# B&R Automation Studio project SDCAxis
Automation Studio 4.5.2.102; Default project; technology packages: Acp10Arnc0 1.0.0

## Configuration Real

CPU 4PP065.0571-P74, AutomationRuntime D4.52, Build 4.1.2, Vc V4.25.0, Safety 1.6

### Task classes (Cpu.sw)
```
Cyclic#1 (cycle 2000 us, tolerance 0 us):
  SDCAxisCtr <- SDCAxisCtrl_X.prg
  SDCAxisCt2 <- SDCAxisCtrl_Z.prg
  SDCAxisCt1 <- SDCAxisCtrl_Y.prg
DataObjects: Arnc0sys
NcDataObjects: AxisInit <- AxisInit.dob, gAxis05a <- gAxis05obj.gAxis05a.dob, gAxis03a <- gAxis03obj.gAxis03a.dob, AxisApt <- AxisApt.dob, gAxis05i <- gAxis05obj.gAxis05i.dob, gAxis03i <- gAxis03obj.gAxis03i.dob, CncInit <- CncInit.dob, CncProg <- CncProg.dob, gmcipvar <- GmcIpUserConfig.gmcipvar.dob, gmcipfun <- GmcIpUserConfig.gmcipfun.dob, gmcipfub <- GmcIpUserConfig.gmcipfub.dob, gmcipubr <- GmcIpUserConfig.gmcipubr.dob, gmcipusm <- GmcIpUserConfig.gmcipusm.dob, gmcipui <- GmcIpUserConfig.gmcipui.dob, gmcipus <- GmcIpUserConfig.gmcipus.dob, gmcipuc <- GmcIpUserConfig.gmcipuc.dob, gmcipsys <- GmcIpConfig.gmcipsys.dob, gmciplbr <- GmcIpConfig.gmciplbr.dob, gmcipcbr <- GmcIpConfig.gmcipcbr.dob, gmciplsm <- GmcIpConfig.gmciplsm.dob, gmcipcsm <- GmcIpConfig.gmcipcsm.dob, gmcipcfg <- GmcIpConfig.gmcipcfg.dob, gmcipiec <- GmcIpConfig.gmcipiec.dob, gmciplog <- GmcIpConfig.gmciplog.dob, gmcipesm <- GmcIpConfig.gmcipesm.dob, gmcipmxd <- GmcIpConfig.gmcipmxd.dob, gmcipmx <- GmcIpConfig.gmcipmx.dob
Binaries: TCData, udbdef, ashwac, ashwd, asfw, iomap, sysconf, Role, User, arconfig, Arnc0map, arnc0cfg, Acp10map, acp10cfg, Acp10map1
Libraries: Acp10sdc, Library, Acp10man, Acp10_MC, sys_lib, brsystem, asstring, AsMath, Arnc0man, DataObj, AsArLog, FileIO, AsArProf, AsMem, Runtime, astime, Acp10par, NcGlobal, powerlnk, asiotime, asieccon
```

### Hardware
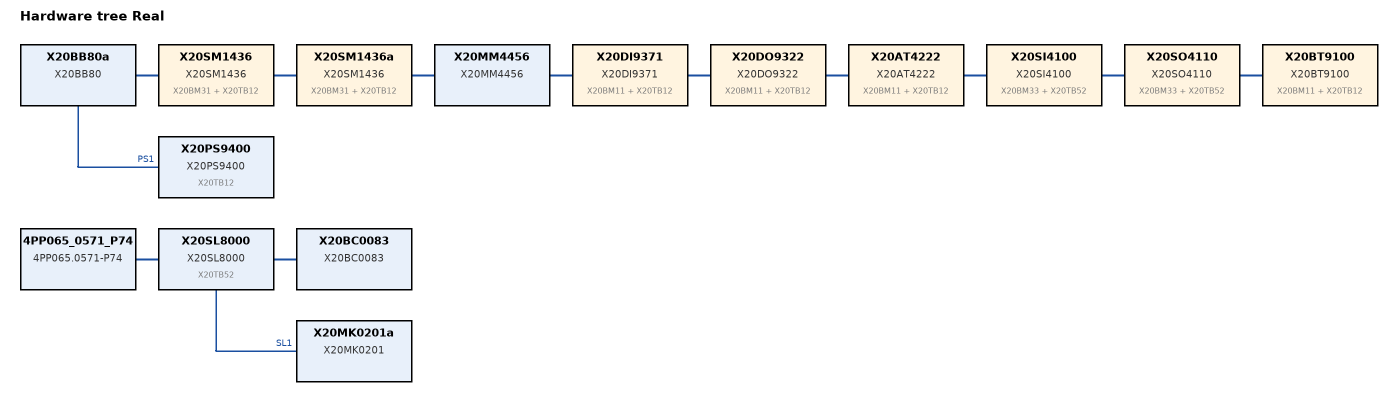
```
4PP065_0571_P74 : 4PP065.0571-P74 v1.1.2.0
  Connector IF4:
    EplInterfaceRedundant = 0
    EplEthInterfaceRedundant = 0
  Connector IF5:
    ActivateDevice = 1
    Mode = Manual
    InternetAddress = 10.0.1.14
    SubnetMask = 255.255.255.0
  ConfigurationID = labBR
  TimerDeviceType = EPLX2X
  TimerDevice = 4PP065_0571_P74.IF4
  TaskClassIdleTime = 2000
  Cyclic1Duration = 2000
  Cyclic1Tolerance = 0
  Cyclic1Output = 1
  Cyclic3Tolerance = 0
  VcObjectName = Visu
X20AT4222 : X20AT4222 v1.2.3.0  [SS1 -> X20TB12f.SS; SL -> X20BM11c.SL1]
X20BB80a : X20BB80 v1.0.2.0
X20BC0083 : X20BC0083 v2.7.0.0  [PLK1 -> X20SL8000.PLK2 (NodeNumber=2) [Cable Type=PowerlinkCable, Length=10, Version=1.0.0.2]; SL -> X20BB80a.SL1]
X20BM11a : X20BM11 v1.0.0.1  [X2X1 -> X20MM4456.X2X2]
X20BM11b : X20BM11 v1.0.0.1  [X2X1 -> X20BM11a.X2X2]
X20BM11c : X20BM11 v1.0.0.1  [X2X1 -> X20BM11b.X2X2]
X20BM11d : X20BM11 v1.0.0.1  [X2X1 -> X20BM33b.X2X2]
X20BM31a : X20BM31 v1.0.0.1  [X2X1 -> X20BB80a.IF1]
X20BM31b : X20BM31 v1.0.0.1  [X2X1 -> X20BM31a.X2X2]
X20BM33a : X20BM33 v1.0.0.4  [X2X1 -> X20BM11c.X2X2]
X20BM33b : X20BM33 v1.0.0.4  [X2X1 -> X20BM33a.X2X2]
X20BT9100 : X20BT9100 v1.0.3.0  [SS1 -> X20TB12g.SS; SL -> X20BM11d.SL1]
X20DI9371 : X20DI9371 v1.0.2.0  [SS1 -> X20TB12d.SS; SL -> X20BM11a.SL1]
X20DO9322 : X20DO9322 v1.0.3.0  [SS1 -> X20TB12e.SS; SL -> X20BM11b.SL1]
X20MK0201a : X20MK0201 v1.0.0.0  [SL -> X20SL8000.SL1]
X20MM4456 : X20MM4456 v1.1.5.0  [X2X1 -> X20BM31b.X2X2]
X20PS9400 : X20PS9400 v1.0.2.4  [SS1 -> X20TB12b.SS; PS -> X20BB80a.PS1]
X20SI4100 : X20SI4100 v1.10.1.1  [SS1 -> X20TB52b.SS; SL -> X20BM33a.SL1]
X20SL8000 : X20SL8000 v1.6.5.1  [PLK1 -> 4PP065_0571_P74.IF4 (NodeNumber=1) [Cable Type=PowerlinkCable, Length=10, Version=1.0.0.2]; PLK2 -> X20BC0083.PLK1 (NodeNumber=1) [Cable Type=PowerlinkCable, Length=10, Version=1.0.0.2]; SS1 -> X20TB52a.SS]
  SafeProject = SafeLOGIC-1
X20SM1436 : X20SM1436 v1.4.2.1  [SS1 -> X20TB12a.SS; SL -> X20BM31a.SL1]
X20SM1436a : X20SM1436 v1.4.2.1  [SS1 -> X20TB12c.SS; SL -> X20BM31b.SL1]
X20SO4110 : X20SO4110 v1.10.1.1  [SS1 -> X20TB52c.SS; SL -> X20BM33b.SL1]
  SafeLogicID = 2
  SafeModuleID = 3
X20TB12a : X20TB12 v1.0.0.0
X20TB12b : X20TB12 v1.0.0.0
X20TB12c : X20TB12 v1.0.0.0
X20TB12d : X20TB12 v1.0.0.0
X20TB12e : X20TB12 v1.0.0.0
X20TB12f : X20TB12 v1.0.0.0
X20TB12g : X20TB12 v1.0.0.0
X20TB52a : X20TB52 v1.0.0.1
X20TB52b : X20TB52 v1.0.0.1
X20TB52c : X20TB52 v1.0.0.1
```

### IoMap.iom - 4PP065_0571_P74/IoMap.iom
```iecst
VAR_CONFIG
	::SDCAxisCtr:pwm_period AT %QW."X20MM4456".PeriodDurationPWM;
	::SDCAxisCtr:coil_pwm_value AT %QW."X20MM4456".PulseWidthCurrentPWM04;
	::SDCAxisCtr:axis_X.pwm_value AT %QW."X20MM4456".PulseWidthCurrentPWM01;
	::SDCAxisCtr:axis_X.reset_error AT %QX."X20MM4456".ClearError01;
	::SDCAxisCtr:axis_X.reset_counter AT %QX."X20MM4456".ResetCounter01;
	::SDCAxisCtr:axis_X.counter AT %IW."X20MM4456".Counter01;
	::SDCAxisCtr:axis_X.endswitch_a_reached AT %IX."X20MM4456".StatusInput03;
	::SDCAxisCtr:axis_X.endswitch_b_reached AT %IX."X20MM4456".StatusInput04;
	::SDCAxisCtr:coil_powered_X AT %IX."X20DI9371".DigitalInput02;
	::SDCAxisCt1:coil_powered_Y AT %IX."X20DI9371".DigitalInput03;
	::SDCAxisCt2:coil_powered_Z AT %IX."X20DI9371".DigitalInput04;
	::SDCAxisCt1:gaxis03.pwm_value AT %QW."X20MM4456".PulseWidthCurrentPWM02;
	::SDCAxisCt1:gaxis03.reset_error AT %QX."X20MM4456".ClearError02;
	::SDCAxisCt1:gaxis03.reset_counter AT %QX."X20MM4456".ResetCounter02;
	::SDCAxisCt1:gaxis03.counter AT %IW."X20MM4456".Counter02;
	::SDCAxisCt1:gaxis03.endswitch_a_reached AT %IX."X20MM4456".StatusInput07;
	::SDCAxisCt1:gaxis03.endswitch_b_reached AT %IX."X20MM4456".StatusInput08;
	::SDCAxisCt2:gaxis05.pwm_value AT %QW."X20MM4456".PulseWidthCurrentPWM03;
	::SDCAxisCt2:gaxis05.reset_error AT %QX."X20MM4456".ClearError03;
	::SDCAxisCt2:gaxis05.reset_counter AT %QX."X20MM4456".ResetCounter03;
	::SDCAxisCt2:gaxis05.counter AT %IW."X20MM4456".Counter03;
	::SDCAxisCt2:gaxis05.endswitch_a_reached AT %IX."X20MM4456".StatusInput11;
	::SDCAxisCt2:gaxis05.endswitch_b_reached AT %IX."X20MM4456".StatusInput12;
END_VAR
```

### Acp10cfg.ncc - 4PP065_0571_P74/Motion/Acp10cfg.ncc
```
NcConfiguration (Version=3.13.1, NcSwId=Acp10)
  ACP10CF1_typ:
    cnt_nettrc_rec_drive = 1500
    bufsize_trace_upload = 1200
    tc_nc_man_task = Cyclic #1
    glob_pv_as_ncobject = Yes
    ncsys_dl_broadcast = Yes
    ncsys_dl_acp_reset = Yes
    safemc_log_err_to_ax = Yes
    network_init:
      ncsw_init_execute = Yes
      automatic_execute = No
      node_nr_warning = Yes
      net_err_before_ncact = Yes
    nettrc:
      enter_parsecrec = Yes
      enter_ncaction = Yes
      save_ring_startidx = Yes
    cam_prof_download:
      cam_dat_dl_parallel = No
      tc_cam_dl_parallel = Task class for NC Manager task
    sdc_if[0]:
      if_name = SDC_IF1
      mc_broadcast_size = 800
      mc_broadcast_extdat = No
```

### Acp10map.ncm - 4PP065_0571_P74/Motion/Acp10map.ncm
```
NcMapping (NcSwId=Acp10, DisabledNodesAreHidden=False)
```

### Acp10map1.ncm - 4PP065_0571_P74/Motion/Acp10map1.ncm
```
NcMapping (NcSwId=ACP10, DisabledNodesAreHidden=False)
  NcObject AxisX (ModuleAddress=SDC_IF1.ST1, InterfaceType=SDC, Type=ncAXIS, Channel=1, AcoposSimulation=Off, InitParameter=AxisInit, AcoposParameter=gAxis03a, AdditionalData=CNC_Enabled="1" , Disabled=FALSE, ModuleDisabled=FALSE)
  NcObject gAxis03 (ModuleAddress=SDC_IF1.ST2, InterfaceType=SDC, Type=ncAXIS, Channel=1, AcoposSimulation=Off, InitParameter=AxisInit, AcoposParameter=gAxis03a, AdditionalData=CNC_Enabled="1", Disabled=FALSE)
  NcObject gAxis05 (ModuleAddress=SDC_IF1.ST3, InterfaceType=SDC, Type=ncAXIS, Channel=1, AcoposSimulation=Off, InitParameter=AxisInit, AcoposParameter=gAxis03a, AdditionalData=CNC_Enabled="1" , Disabled=FALSE)
```

### Arnc0cfg.ncc - 4PP065_0571_P74/Motion/Arnc0cfg.ncc
```
NcConfiguration (Version=3.13.0, NcSwId=Arnc0)
  ARNC0CFG_typ:
    sampling_rate = 2000
    cnt_nettrc_rec_drive = 150
    bufsize_sys_trace = 16#00005000
    enable_mp_log = Yes
    tc_nc_man_task = Cyclic #1
    bg_load = 1
    glob_pv_as_ncobject = Yes
```

### Arnc0map.ncm - 4PP065_0571_P74/Motion/Arnc0map.ncm
```
NcMapping (NcSwId=Arnc0, DisabledNodesAreHidden=True)
  NcObject CNCsys (Type=ncCNCSYS, Channel=1, AcoposSimulation=Off, InitParameter=CncInit, Disabled=FALSE, ModuleDisabled=FALSE)
  NcObject CNC2 (Type=ncCNCSYS, Channel=2, AcoposSimulation=Off, Disabled=TRUE, ModuleDisabled=FALSE)
  NcObject CNC3 (Type=ncCNCSYS, Channel=3, AcoposSimulation=Off, Disabled=TRUE, ModuleDisabled=FALSE)
  NcObject CNC4 (Type=ncCNCSYS, Channel=4, AcoposSimulation=Off, Disabled=TRUE, ModuleDisabled=FALSE)
  NcObject CNC5 (Type=ncCNCSYS, Channel=5, AcoposSimulation=Off, Disabled=TRUE, ModuleDisabled=FALSE)
  NcObject CNC6 (Type=ncCNCSYS, Channel=6, AcoposSimulation=Off, Disabled=TRUE, ModuleDisabled=FALSE)
  NcObject CNC7 (Type=ncCNCSYS, Channel=7, AcoposSimulation=Off, Disabled=TRUE, ModuleDisabled=FALSE)
  NcObject CNC8 (Type=ncCNCSYS, Channel=8, AcoposSimulation=Off, Disabled=TRUE, ModuleDisabled=FALSE)
  NcObject CNC9 (Type=ncCNCSYS, Channel=9, AcoposSimulation=Off, Disabled=TRUE, ModuleDisabled=FALSE)
  NcObject CNC10 (Type=ncCNCSYS, Channel=10, AcoposSimulation=Off, Disabled=TRUE, ModuleDisabled=FALSE)
  NcObject CNC11 (Type=ncCNCSYS, Channel=11, AcoposSimulation=Off, Disabled=TRUE, ModuleDisabled=FALSE)
  NcObject CNC12 (Type=ncCNCSYS, Channel=12, AcoposSimulation=Off, Disabled=TRUE, ModuleDisabled=FALSE)
  NcObject CNC13 (Type=ncCNCSYS, Channel=13, AcoposSimulation=Off, Disabled=TRUE, ModuleDisabled=FALSE)
  NcObject CNC14 (Type=ncCNCSYS, Channel=14, AcoposSimulation=Off, Disabled=TRUE, ModuleDisabled=FALSE)
  NcObject CNC15 (Type=ncCNCSYS, Channel=15, AcoposSimulation=Off, Disabled=TRUE, ModuleDisabled=FALSE)
  NcObject CNC16 (Type=ncCNCSYS, Channel=16, AcoposSimulation=Off, Disabled=TRUE, ModuleDisabled=FALSE)
  NcObject CNC17 (Type=ncCNCSYS, Channel=17, AcoposSimulation=Off, Disabled=TRUE, ModuleDisabled=FALSE)
  NcObject CNC18 (Type=ncCNCSYS, Channel=18, AcoposSimulation=Off, Disabled=TRUE, ModuleDisabled=FALSE)
  NcObject CNC19 (Type=ncCNCSYS, Channel=19, AcoposSimulation=Off, Disabled=TRUE, ModuleDisabled=FALSE)
  NcObject CNC20 (Type=ncCNCSYS, Channel=20, AcoposSimulation=Off, Disabled=TRUE, ModuleDisabled=FALSE)
  NcObject CNC21 (Type=ncCNCSYS, Channel=21, AcoposSimulation=Off, Disabled=TRUE, ModuleDisabled=FALSE)
  NcObject CNC22 (Type=ncCNCSYS, Channel=22, AcoposSimulation=Off, Disabled=TRUE, ModuleDisabled=FALSE)
  NcObject CNC23 (Type=ncCNCSYS, Channel=23, AcoposSimulation=Off, Disabled=TRUE, ModuleDisabled=FALSE)
  NcObject CNC24 (Type=ncCNCSYS, Channel=24, AcoposSimulation=Off, Disabled=TRUE, ModuleDisabled=FALSE)
```

## Configuration Simulation

CPU , AutomationRuntime J4.25, Safety 1.10

### Task classes (Cpu.sw)
```
Cyclic#1 (cycle 2000 us, tolerance 0 us):
  SDCAxisCtr <- SDCAxisCtrl_X.prg
  ncsdcctrl <- ncsdcctrl.prg
DataObjects: Acp10sys
NcDataObjects: AxisApt <- AxisApt.dob, AxisInit <- AxisInit.dob, acp10etxen <- acp10etxen.dob, gAxis05a <- gAxis05obj.gAxis05a.dob, gAxis05i <- gAxis05obj.gAxis05i.dob
Binaries: TCData, ashwd, sysconf, asfw, arconfig, iomap, Acp10map, Acp10map1, arnc0cfg, acp10cfg
Libraries: AsIecCon, astime, Acp10sdc, Acp10man, Acp10par, NcGlobal, asstring, AsIOTime, Acp10_MC, brsystem, sys_lib, Runtime, Acp10sim, fileio, powerlnk, Library, AsBrStr
```

### Hardware
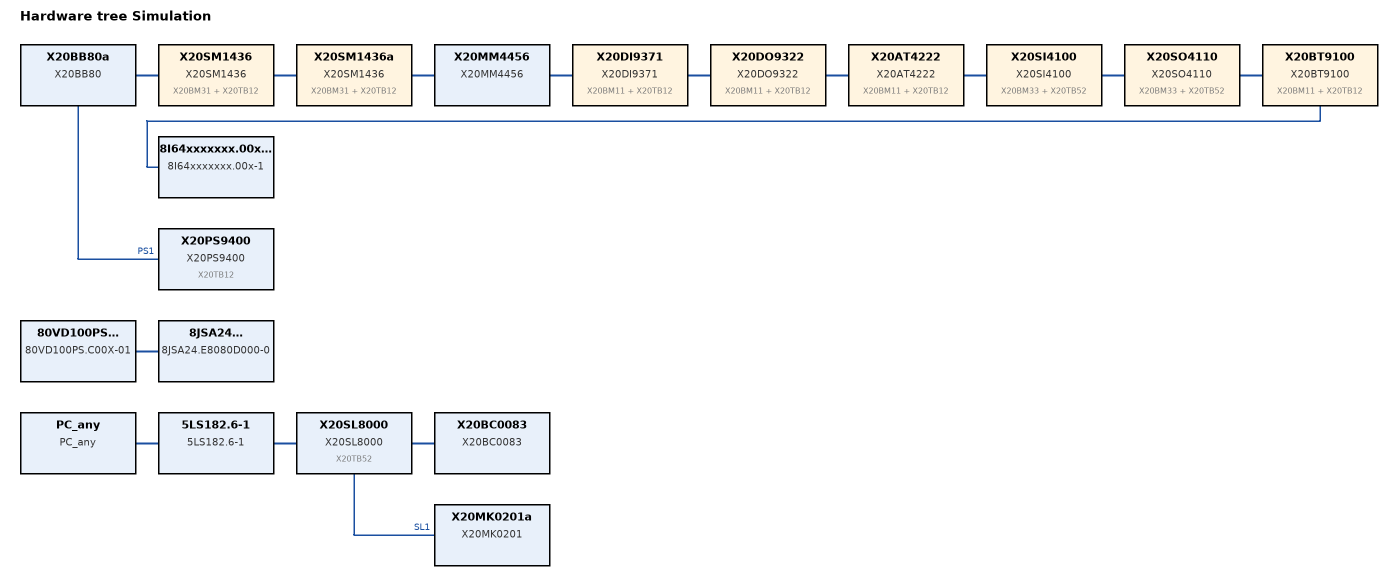
```
5LS182.6-1 : 5LS182.6-1 v1.3.0.0  [SL -> PC_any.SL1]
80VD100PS.C00X-01 : 80VD100PS.C00X-01 v2.3.0.1
8I64xxxxxxx.00x-1 : 8I64xxxxxxx.00x-1 v1.3.9.1  [X2X1 -> X20BT9100.X2X1 [Cable Type=X2XCable, Length=10, Version=1.0.0.2]]
  BothEndSwitchesAreNormallyOpen_r1 = on
  QuickStopIsNormallyOpen_r1 = on
8JSA24.E8080D000-0 : 8JSA24.E8080D000-0 v1.0.6.30  [MT -> 80VD100PS.C00X-01.MT1]
PC_any : PC_any v1.1.0.0 (OrderNumber=PC)
  ConfigurationID = SDCAxis_Simulation
  SystemTick = 2000
  Cyclic1Duration = 2000
  Cyclic1Tolerance = 0
  Cyclic1Output = 1
X20AT4222 : X20AT4222 v1.2.3.0  [SS1 -> X20TB12f.SS; SL -> X20BM11c.SL1]
X20BB80a : X20BB80 v1.0.2.0
X20BC0083 : X20BC0083 v2.7.0.0  [PLK2 -> X20SL8000.PLK2 (NodeNumber=2) [Cable Type=PowerlinkCable, Length=10, Version=1.0.0.2]; SL -> X20BB80a.SL1]
X20BM11a : X20BM11 v1.0.0.1  [X2X1 -> X20MM4456.X2X2]
X20BM11b : X20BM11 v1.0.0.1  [X2X1 -> X20BM11a.X2X2]
X20BM11c : X20BM11 v1.0.0.1  [X2X1 -> X20BM11b.X2X2]
X20BM11d : X20BM11 v1.0.0.1  [X2X1 -> X20BM33b.X2X2]
X20BM31a : X20BM31 v1.0.0.1  [X2X1 -> X20BB80a.IF1]
X20BM31b : X20BM31 v1.0.0.1  [X2X1 -> X20BM31a.X2X2]
X20BM33a : X20BM33 v1.0.0.4  [X2X1 -> X20BM11c.X2X2]
X20BM33b : X20BM33 v1.0.0.4  [X2X1 -> X20BM33a.X2X2]
X20BT9100 : X20BT9100 v1.0.3.0  [SS1 -> X20TB12g.SS; SL -> X20BM11d.SL1]
X20DI9371 : X20DI9371 v1.0.2.0  [SS1 -> X20TB12d.SS; SL -> X20BM11a.SL1]
X20DO9322 : X20DO9322 v1.0.3.0  [SS1 -> X20TB12e.SS; SL -> X20BM11b.SL1]
X20MK0201a : X20MK0201 v1.0.0.0  [SL -> X20SL8000.SL1]
X20MM4456 : X20MM4456 v1.1.5.0  [X2X1 -> X20BM31b.X2X2]
X20PS9400 : X20PS9400 v1.0.2.4  [SS1 -> X20TB12b.SS; PS -> X20BB80a.PS1]
X20SI4100 : X20SI4100 v1.10.1.1  [SS1 -> X20TB52b.SS; SL -> X20BM33a.SL1]
X20SL8000 : X20SL8000 v1.6.5.1  [PLK1 -> 5LS182.6-1.IF1 (NodeNumber=1) [Cable Type=PowerlinkCable, Length=10, Version=1.0.0.2]; PLK2 -> X20BC0083.PLK2 (NodeNumber=1) [Cable Type=PowerlinkCable, Length=10, Version=1.0.0.2]; SS1 -> X20TB52a.SS]
  SafeProject = SafeLOGIC-1
X20SM1436 : X20SM1436 v1.4.2.1  [SS1 -> X20TB12a.SS; SL -> X20BM31a.SL1]
X20SM1436a : X20SM1436 v1.4.2.1  [SS1 -> X20TB12c.SS; SL -> X20BM31b.SL1]
X20SO4110 : X20SO4110 v1.10.1.1  [SS1 -> X20TB52c.SS; SL -> X20BM33b.SL1]
  SafeLogicID = 2
  SafeModuleID = 3
X20TB12a : X20TB12 v1.0.0.0
X20TB12b : X20TB12 v1.0.0.0
X20TB12c : X20TB12 v1.0.0.0
X20TB12d : X20TB12 v1.0.0.0
X20TB12e : X20TB12 v1.0.0.0
X20TB12f : X20TB12 v1.0.0.0
X20TB12g : X20TB12 v1.0.0.0
X20TB52a : X20TB52 v1.0.0.1
X20TB52b : X20TB52 v1.0.0.1
X20TB52c : X20TB52 v1.0.0.1
```

### IOMap.iom - PC_any/IOMap.iom
```iecst
VAR_CONFIG
	::SDCAxisCtr:pwm_period AT %QW."X20MM4456".PeriodDurationPWM;
	::SDCAxisCtr:coil_pwm_value AT %QW."X20MM4456".PulseWidthCurrentPWM04;
	::SDCAxisCtr:axis_X.pwm_value AT %QW."X20MM4456".PulseWidthCurrentPWM01;
	::SDCAxisCtr:axis_X.reset_error AT %QX."X20MM4456".ClearError01;
	::SDCAxisCtr:axis_X.reset_counter AT %QX."X20MM4456".ResetCounter01;
	::SDCAxisCtr:axis_X.counter AT %IW."X20MM4456".Counter01;
	::SDCAxisCtr:axis_X.endswitch_a_reached AT %IX."X20MM4456".StatusInput03; (*Logical condition input 01=Motor 01:A*)
	::SDCAxisCtr:axis_X.endswitch_b_reached AT %IX."X20MM4456".StatusInput04; (*Logical condition input 02=Motor 01:B*)
	::SDCAxisCtr:coil_powered AT %IX."X20DI9371".DigitalInput01;
	Cyclic#1.gAxis03_DrvIf.iLifeCnt AT %IB."8I64xxxxxxx.00x-1".SDC_LifeCnt;
	Cyclic#1.gAxis03_DrvIf.iDrvOK AT %IX."8I64xxxxxxx.00x-1".ETAD_Input_Bool_02;
	Cyclic#1.gAxis03_DrvIf.oSetTime AT %QW."8I64xxxxxxx.00x-1".SDC_SetTime;
	Cyclic#1.gAxis03_DrvIf.oSetPos AT %QW."8I64xxxxxxx.00x-1".LFRD_Output;
	Cyclic#1.gAxis03_DiDoIf.iLifeCntDriveReady AT %IB."8I64xxxxxxx.00x-1".SDC_LifeCnt;
	Cyclic#1.gAxis03_DiDoIf.iLifeCntDriveEnable AT %IB."8I64xxxxxxx.00x-1".SDC_LifeCnt;
	Cyclic#1.gAxis03_DiDoIf.oDriveEnable AT %QX."8I64xxxxxxx.00x-1".CMDD_Output_Bool_00;
	Cyclic#1.gAxis03_ModuleOk AT %QX."8I64xxxxxxx.00x-1".CMDD_Output_Bool_01;
	Cyclic#1.gAxis03_ModuleOk AT %QX."8I64xxxxxxx.00x-1".CMDD_Output_Bool_02;
	Cyclic#1.gAxis03_ModuleOk AT %IX."8I64xxxxxxx.00x-1".ModuleOk;
	Cyclic#1.gAxis03_DiDoIf.oDriveEnable AT %QX."8I64xxxxxxx.00x-1".CMDD_Output_Bool_03;
	Cyclic#1.gAxis03_DiDoIf.iDriveReady AT %IX."8I64xxxxxxx.00x-1".ETAD_Input_Bool_02;
	      Cyclic#1.gAxis05_DrvIf.iLifeCnt AT %IB."X20SM1436".LifeCnt;
	      Cyclic#1.gAxis05_DrvIf.iDrvOK AT %IX."X20SM1436".DrvOk01;
	      Cyclic#1.gAxis05_DrvIf.oBoostCurrent AT %QX."X20SM1436".BoostCurrent01;
	      Cyclic#1.gAxis05_DrvIf.oStandStillCurrent AT %QX."X20SM1436".StandstillCurrent01;
	      Cyclic#1.gAxis05_DrvIf.oSetTime AT %QW."X20SM1436".SetTime01;
	      Cyclic#1.gAxis05_MotorStep0 AT %QW."X20SM1436".Motor1Step0;
	      Cyclic#1.gAxis05_DiDoIf.iLifeCntDriveEnable AT %IB."X20SM1436".LifeCnt;
	      Cyclic#1.gAxis05_DiDoIf.iLifeCntDriveReady AT %IB."X20SM1436".LifeCnt;
	      Cyclic#1.gAxis05_DiDoIf.iDriveReady AT %IX."X20SM1436".DrvOk01;
	      Cyclic#1.gAxis05_DiDoIf.oDriveEnable AT %QX."X20SM1436".DriveEnable01;
	      Cyclic#1.gAxis05_EncIf1.iLifeCnt AT %IB."X20SM1436".LifeCnt;
	      Cyclic#1.gAxis05_EncIf1.iEncOK AT %IX."X20SM1436".EncOk01;
	      Cyclic#1.gAxis05_EncIf1.iActPos AT %IW."X20SM1436".ActPos01;
	      Cyclic#1.gAxis05_EncIf1.iRefPulsePos AT %IW."X20SM1436".RefPulsePos01;
	      Cyclic#1.gAxis05_EncIf1.iRefPulseCnt AT %IB."X20SM1436".RefPulseCnt01;
	      Cyclic#1.gAxis05_EncIf1.iActTime AT %IW."X20SM1436".ActTime01;
END_VAR
```

### Acp10cfg.ncc - PC_any/Motion/Acp10cfg.ncc
```
NcConfiguration (Version=3.13.1, NcSwId=Acp10)
  ACP10CF1_typ:
    cnt_nettrc_rec_drive = 150
    bufsize_trace_upload = 1200
    tc_nc_man_task = Cyclic #1
    glob_pv_as_ncobject = Yes
    ncsys_dl_broadcast = Yes
    ncsys_dl_acp_reset = Yes
    safemc_log_err_to_ax = Yes
    network_init:
      ncsw_init_execute = Yes
      automatic_execute = No
      node_nr_warning = Yes
      net_err_before_ncact = Yes
    nettrc:
      enter_parsecrec = Yes
      enter_ncaction = Yes
      save_ring_startidx = No
    cam_prof_download:
      cam_dat_dl_parallel = No
      tc_cam_dl_parallel = Task class for NC Manager task
    sdc_if[0]:
      if_name = SDC_IF1
      mc_broadcast_size = 800
      mc_broadcast_extdat = No
```

### Acp10map.ncm - PC_any/Motion/Acp10map.ncm
```
NcMapping (NcSwId=Acp10)
  NcObject gAxis04 (ModuleId=8I64xxxxxxx.00x-1, ModuleAddress=SDC_IF1.ST2, Type=ncAXIS, Channel=1, AcoposSimulation=Off, InitParameter=gAxis03i, AcoposParameter=gAxis03a, AdditionalData=CNC_Enabled="1" , Disabled=FALSE, ModuleDisabled=FALSE)
  NcObject gAxis05 (ModuleId=X20SM1436, ModuleAddress=SDC_IF1.ST3, Type=ncAXIS, Channel=1, AcoposSimulation=Off, InitParameter=gAxis05i, AcoposParameter=gAxis05a, Disabled=FALSE, ModuleDisabled=FALSE)
  NcObject X20SM1436a_ncAXIS1 (ModuleId=X20SM1436a, ModuleAddress=SDC_IF1.ST4, Type=ncAXIS, Channel=1, AcoposSimulation=Off, Disabled=TRUE, ModuleDisabled=FALSE)
```

### Acp10map1.ncm - PC_any/Motion/Acp10map1.ncm
```
NcMapping (NcSwId=ACP10, DisabledNodesAreHidden=False)
  NcObject MyLittleAxis (ModuleAddress=SDC_IF1.ST1, InterfaceType=SDC, Type=ncAXIS, Channel=1, AcoposSimulation=Off, InitParameter=MyLittleIn, AcoposParameter=MyLittleAp, Disabled=FALSE, ModuleDisabled=FALSE)
```

### Arnc0cfg.ncc - PC_any/Motion/Arnc0cfg.ncc
```
NcConfiguration (Version=1.45.0, NcSwId=ARNC0)
  ARNC0CFG_typ:
    sampling_rate = 4000
    cnt_nettrc_rec_drive = 150
    bufsize_sys_trace = 16#00005000
    enable_mp_log = Yes
    tc_nc_man_task = Cyclic #1
    bg_load = 1
    glob_pv_as_ncobject = Yes
```

## Logical view

Binary libraries used (declarations not repeated): Runtime, Operator, AsIecCon, astime, Acp10sdc 3.13.1, Acp10man 3.13.1, Acp10par 3.13.1, NcGlobal 3.13.1, asstring, AsIOTime, Acp10_MC 3.13.1, brsystem, sys_lib, Acp10sim 3.13.1, AsMath, Arnc0man 3.13.0, DataObj, AsArLog, FileIO, AsArProf, AsMem, AsBrStr

### Global.var - Global variables
```iecst
VAR
	AxisX : ACP10AXIS_typ := (0);
	AxisX_EncIf : SdcEncIf16_typ := (0);
	AxisX_DrvIf : SdcDrvIf16_typ := (0);
	AxisX_DiDoIf : SdcDiDoIf_typ := (0);
	AxisX_HW : SdcHwCfg_typ := (0);
	gAxis01 : ACP10AXIS_typ := (0);
	gAxis02 : ACP10AXIS_typ := (0);
	gAxisTest : ACP10AXIS_typ := (0);
	New_Variable : USINT := 0;
	gAxisTest_HW : SdcHwCfg_typ := (0);
	gAxis05_EncIf : SdcEncIf16_typ := (0);
	gAxis03_EncIf : SdcEncIf16_typ := (0);
	gAxisTest_DrvIf : SdcDrvIf16_typ := (0);
	gAxisTest_DiDoIf : SdcDiDoIf_typ := (0);
	gAxis03 : ACP10AXIS_typ := (0);
	gAxis03_HW : SdcHwCfg_typ := (0);
	gAxis03_DrvIf : SdcDrvIf16_typ := (0);
	gAxis03_DiDoIf : SdcDiDoIf_typ := (0);
	CNCsys : ARNC0CNC_typ;
	gAxis04 : ACP10AXIS_typ := (0);
	gAxis05 : ACP10AXIS_typ := (0);
	gAxis05_HW : SdcHwCfg_typ := (0);
	gAxis05_DrvIf : SdcDrvIf16_typ := (0);
	gAxis05_DiDoIf : SdcDiDoIf_typ := (0);
	gAxis05_MotorStep0 : INT := 0;
	coil_powered : BOOL := FALSE;
	coil_pwm_value : INT := 0;
	fb_regulator : FB_Regulator;
	pwm_period : UINT := 0;
	axis_X : FB_Axis := (0);
	iPosHwEnd : BOOL := FALSE;
	iNegHwEnd : BOOL := FALSE;
	iActPos : USINT := 0;
	oSetPos : USINT := 0;
END_VAR
```

### Package Logical/Libraries - Global libraries

### Library Logical/Libraries/Library (ANSIC)

#### Library.fun
```iecst
FUNCTION_BLOCK FB_Motor (*TODO: Add your comment here*) (*$GROUP=User,$CAT=User,$GROUPICON=User.png,$CATICON=User.png*)
	VAR_INPUT
		in : REAL;
	END_VAR
	VAR_OUTPUT
		out_w : REAL;
		out_phi : REAL;
	END_VAR
	VAR
		k_e : REAL;
		T_m : REAL;
		dt : REAL;
		integrator : FB_Integrator;
		integrator_phi : FB_Integrator;
	END_VAR
END_FUNCTION_BLOCK

FUNCTION_BLOCK FB_Integrator (*TODO: Add your comment here*) (*$GROUP=User,$CAT=User,$GROUPICON=User.png,$CATICON=User.png*)
	VAR_INPUT
		in : REAL;
		dt : REAL;
	END_VAR
	VAR_OUTPUT
		out : REAL;
	END_VAR
	VAR
		state : REAL := 0.0;
	END_VAR
END_FUNCTION_BLOCK

FUNCTION_BLOCK FB_Controller (* *) (*$GROUP=User,$CAT=User,$GROUPICON=User.png,$CATICON=User.png*)
	VAR_INPUT
		in : REAL;
	END_VAR
	VAR_OUTPUT
		out : REAL;
	END_VAR
	VAR
		k_i : REAL;
		sum : REAL;
		k_p : REAL;
		dt : REAL;
		max_abs_value : REAL;
		integrator : FB_Integrator;
		last_sum : REAL;
	END_VAR
END_FUNCTION_BLOCK

FUNCTION_BLOCK FB_Endswitch (*TODO: Add your comment here*) (*$GROUP=User,$CAT=User,$GROUPICON=User.png,$CATICON=User.png*)
	VAR_INPUT
		in : REAL;
		neg_value : REAL;
		pos_value : REAL;
	END_VAR
	VAR_OUTPUT
		neg_reached : BOOL;
		pos_reached : BOOL;
	END_VAR
END_FUNCTION_BLOCK

FUNCTION_BLOCK FB_Axis (*TODO: Add your comment here*) (*$GROUP=User,$CAT=User,$GROUPICON=User.png,$CATICON=User.png*)
	VAR_INPUT
		u : REAL;
		reset_error : BOOL;
		endswitch_a_reached : BOOL;
		endswitch_b_reached : BOOL;
		pwm_percentage : SINT;
	END_VAR
	VAR_OUTPUT
		reset_counter : BOOL;
		pwm_value : INT;
	END_VAR
	VAR_OUTPUT RETAIN
		counter : INT;
	END_VAR
	VAR_OUTPUT
		speed : REAL;
	END_VAR
	VAR
		i : INT;
		last_counter : INT;
		dir : BOOL;
		spid : REAL;
		k : INT;
	END_VAR
END_FUNCTION_BLOCK

{REDUND_ERROR} FUNCTION_BLOCK FB_Regulator (*TODO: Add your comment here*) (*$GROUP=User,$CAT=User,$GROUPICON=User.png,$CATICON=User.png*)
	VAR_INPUT
		e : REAL;
	END_VAR
	VAR_OUTPUT
		u : REAL;
	END_VAR
	VAR
		k_p : REAL;
		k_i : REAL;
		integrator : FB_Integrator;
		iyOld : REAL;
		max_abc_value : REAL := 24;
		dt : REAL;
		x : REAL;
	END_VAR
END_FUNCTION_BLOCK
```

#### FB_Motor.c
```c
#include <bur/plctypes.h>
#ifdef __cplusplus
	extern "C"
	{
#endif
	#include "Library.h"
#ifdef __cplusplus
	};
#endif
/* TODO: Add your comment here */
void FB_Motor(struct FB_Motor* inst)
{/*
	inst->integrator.in = (inst->u/inst->ke - inst->w) * (inst->dt/inst->Tm);
	FB_Integrator(&inst->integrator);
	inst->w = inst->integrator.out;
	inst->integrator.in = inst->w * inst->dt;
	FB_Integrator(&inst->integrator);
	inst->phi = inst->integrator.out;*/
}
```

#### FB_Controller.c
```c
#include <bur/plctypes.h>
#ifdef __cplusplus
	extern "C"
	{
#endif
	#include "Library.h"
#ifdef __cplusplus
	};
#endif

void FB_Controller(struct FB_Controller* inst)
{

}
```

#### FB_Integrator.c
```c
#include <bur/plctypes.h>
#ifdef __cplusplus
	extern "C"
	{
#endif
	#include "Library.h"
#ifdef __cplusplus
	};
#endif
/* TODO: Add your comment here */
void FB_Integrator(struct FB_Integrator* inst)
{
	inst->out = inst->dt * inst->in + inst->state;
	inst->state = inst->out;
}
```

#### FB_Endswitch.c
```c
#include <bur/plctypes.h>
#ifdef __cplusplus
	extern "C"
	{
#endif
	#include "Library.h"
#ifdef __cplusplus
	};
#endif
/* TODO: Add your comment here */
void FB_Endswitch(struct FB_Endswitch* inst)
{

}
```

#### FB_Axis.c
```c
#include <bur/plctypes.h>
#ifdef __cplusplus
	extern "C"
	{
#endif
	#include "Library.h"
#ifdef __cplusplus
	};
#endif
/* TODO: Add your comment here */
void FB_Axis(struct FB_Axis* inst)
{
	/*if (inst->endswitch_a_reached == 1 )
	{
		inst->dir = 1;
	}
	if (inst->endswitch_b_reached == 1 )
	{
		inst->dir = 0;
	}

	if(inst->dir == 1)
	{
		//inst->reset_counter = 0;
		inst->u = -inst->u;
		inst->pwm_value = (inst->u/24.0) * 32767;
	}
	if(inst->dir == 0)
	{*/
		//inst->reset_counter = 0;
		inst->pwm_value = (inst->u/24.0) * 32767;
//	}
	if (inst->i == 1000)
	{
		inst->speed = (inst->counter - inst->last_counter)/2;
		inst->last_counter = inst->counter;
		inst->i = 0;
	}
	inst->spid = inst->speed;
	inst->i++;
}
```

#### FB_Regulator.c
```c
#include <bur/plctypes.h>
#ifdef __cplusplus
	extern "C"
	{
#endif
	#include "Library.h"
#ifdef __cplusplus
	};
#endif
/* TODO: Add your comment here */
void FB_Regulator(struct FB_Regulator* inst)
{
	float BON(float x)
		{
		if(x < 0)
		{
			if(x < -inst->max_abc_value)
				return -inst->max_abc_value;
			else
				return x;
		}
		else
		{
			if(x > inst->max_abc_value)
				return inst->max_abc_value;
			else
				return x;
		}

	}
	inst->integrator.in = inst->e * inst->k_i * inst->dt + inst->iyOld;
	FB_Integrator(&inst->integrator);
	inst->u = BON((BON(inst->e * inst->k_p) + inst->integrator.out));

	inst->iyOld = inst->u - (BON(inst->e * inst->k_p) + inst->integrator.out);
}
```

### Library Logical/Libraries/Library1 (ANSIC)

#### Library1.fun - Exported functions and function blocks
```iecst
{REDUND_ERROR} {REDUND_UNREPLICABLE} FUNCTION_BLOCK FB_Integrator (*TODO: Add your comment here*) (*$GROUP=User,$CAT=User,$GROUPICON=User.png,$CATICON=User.png*)
	VAR_INPUT
		in : {REDUND_UNREPLICABLE} REAL;
	END_VAR
	VAR_OUTPUT
		out : {REDUND_UNREPLICABLE} REAL;
	END_VAR
	VAR
		dt : {REDUND_UNREPLICABLE} REAL;
	END_VAR
END_FUNCTION_BLOCK

{REDUND_ERROR} {REDUND_UNREPLICABLE} FUNCTION_BLOCK FBMotor (*TODO: Add your comment here*) (*$GROUP=User,$CAT=User,$GROUPICON=User.png,$CATICON=User.png*)
	VAR_INPUT
		u : {REDUND_UNREPLICABLE} REAL;
	END_VAR
	VAR_OUTPUT
		w : {REDUND_UNREPLICABLE} REAL;
		phi : {REDUND_UNREPLICABLE} REAL;
	END_VAR
	VAR
		integrator : {REDUND_UNREPLICABLE} FB_Integrator;
		Tm : {REDUND_UNREPLICABLE} REAL;
		ke : {REDUND_UNREPLICABLE} REAL;
		dt : {REDUND_UNREPLICABLE} REAL;
	END_VAR
END_FUNCTION_BLOCK

{REDUND_ERROR} {REDUND_UNREPLICABLE} FUNCTION_BLOCK FB_Regulator (*TODO: Add your comment here*) (*$GROUP=User,$CAT=User,$GROUPICON=User.png,$CATICON=User.png*)
	VAR_INPUT
		e : {REDUND_UNREPLICABLE} REAL;
	END_VAR
	VAR_OUTPUT
		u : {REDUND_UNREPLICABLE} REAL;
	END_VAR
	VAR
		k_p : {REDUND_UNREPLICABLE} REAL;
		k_i : {REDUND_UNREPLICABLE} REAL;
		integrator : {REDUND_UNREPLICABLE} FB_Integrator;
		iyOld : {REDUND_UNREPLICABLE} REAL;
		max_abc_value : {REDUND_UNREPLICABLE} REAL;
		dt : {REDUND_UNREPLICABLE} REAL;
		x : {REDUND_UNREPLICABLE} REAL;
	END_VAR
END_FUNCTION_BLOCK
```

#### FB_Integrator.c
```c
#include <bur/plctypes.h>
#ifdef __cplusplus
	extern "C"
	{
#endif
	#include "Library1.h"
#ifdef __cplusplus
	};
#endif
/* TODO: Add your comment here */
void FB_Integrator(struct FB_Integrator* inst)
{
	inst->out = inst->in  + inst->out;

}
```

#### FBMotor.c
```c
#include <bur/plctypes.h>
#ifdef __cplusplus
	extern "C"
	{
#endif
	#include "Library1.h"
#ifdef __cplusplus
	};
#endif
/* TODO: Add your comment here */
void FBMotor(struct FBMotor* inst)
{
	inst->integrator.in = (inst->u/inst->ke - inst->w) * (inst->dt/inst->Tm);
	FB_Integrator(&inst->integrator);
	inst->w = inst->integrator.out;
	inst->integrator.in = inst->w * inst->dt;
	FB_Integrator(&inst->integrator);
	inst->phi = inst->integrator.out;
}
```

#### FB_Regulator.c
```c
#include <bur/plctypes.h>
#ifdef __cplusplus
	extern "C"
	{
#endif
	#include "Library1.h"
#ifdef __cplusplus
	};
#endif
/* TODO: Add your comment here */
void FB_Regulator(struct FB_Regulator* inst)
{
	float BON(float x)
	{
		if(x < 0)
		{
			if(x < -inst->max_abc_value)
				return -inst->max_abc_value;
			else
				return x;
		}
		else
		{
			if(x > inst->max_abc_value)
				return inst->max_abc_value;
			else
				return x;
		}

	}
	inst->integrator.in = inst->e * inst->k_i * inst->dt + inst->iyOld;
	FB_Integrator(&inst->integrator);
	inst->u = BON((BON(inst->e * inst->k_p) + inst->integrator.out));

	inst->iyOld = inst->u - (BON(inst->e * inst->k_p) + inst->integrator.out);
}
```

### Data object Logical/AxisApt (Apt)

#### AcpParTab.apt
```
AcoposParameterTable:
  Root Parameters:
    64201 = 4000 (Name=SERVO_V_MAX_OUTPUT, Unit=Units/s)  // Servo drive adjustment: Velocity at maximum output value
    109 = 24 (Name=SCALE_ENCOD_INCR)  // Encoder1: Encoder scaling: increments per encoder revolution
```

### Data object Logical/AxisInit (Ax)

#### AxInitAcp10.ax
```
InitParameter (Version=3.13.1, NcSwId=ACP10)
  ACP10AXIS_typ:
    dig_in:
      level:
        reference = ncACTIV_HI
        pos_hw_end = ncACTIV_HI
        neg_hw_end = ncACTIV_HI
        trigger1 = ncACTIV_HI
        trigger2 = ncACTIV_HI
    encoder_if:
      parameter:
        count_dir = ncSTANDARD
        scaling:
          load:
            units = 3000
            rev_motor = 1
    limit:
      parameter:
        v_pos = 7500.0
        v_neg = 7500.0
        a1_pos = 10000.0
        a2_pos = 10000.0
        a1_neg = 10000.0
        a2_neg = 10000.0
        t_jolt = 0.0
        t_in_pos = 0.0
        pos_sw_end = 8388607
        neg_sw_end = -8388608
        ds_warning = 500.0
        ds_stop = 50000.0
        a_stop = 1.0E+30
        dv_stop = 0.0
        dv_stop_mode = ncOFF
    controller:
      mode = ncPOSITION
      position:
        kv = 10.0
        tn = 0.0
        t_predict = 0.04
        t_total = 0.04
        p_max = 10000.0
        i_max = 0.0
      speed:
        kv = 2.0
        tn = 0.0
        t_filter = 0.0
        isq_filter1:
          type = ncOFF
          a0 = 0.0
          a1 = 0.0
          b0 = 0.0
          b1 = 0.0
          b2 = 0.0
          c0_par_id = 0
          c1_par_id = 0
        isq_filter2:
          type = ncOFF
          a0 = 0.0
          a1 = 0.0
          b0 = 0.0
          b1 = 0.0
          b2 = 0.0
          c0_par_id = 0
          c1_par_id = 0
        isq_filter3:
          type = ncOFF
          a0 = 0.0
          a1 = 0.0
          b0 = 0.0
          b1 = 0.0
          b2 = 0.0
          c0_par_id = 0
          c1_par_id = 0
      uf:
        type = ncLINEAR
        auto_config = ncMOTOR_PAR
        u0 = 0.0
        un = 0.0
        fn = 50.0
        k_f_slip = 0.0
      ff:
        torque_load = 0.0
        torque_pos = 0.0
        torque_neg = 0.0
        kv_torque = 0.0
        inertia = 0.0
        t_filter_a = 0.0
    move:
      stop:
        parameter[0]:
          decel_ramp = ncA_LIMIT
          controller = ncON
        parameter[1]:
          decel_ramp = ncA_LIMIT
          controller = ncON
        parameter[2]:
          decel_ramp = ncA_LIMIT
          controller = ncON
        parameter[3]:
          decel_ramp = ncA_LIMIT
          controller = ncON
        quickstop:
          decel_ramp = ncA_LIMIT
        drive_error:
          decel_ramp = ncA_LIMIT
      homing:
        parameter:
          s = 0
          v_switch = 6000.0
          v_trigger = 2000.0
          a = 10000.0
          mode = ncEND_SWITCH
          edge_sw = ncNEGATIVE
          start_dir = ncPOSITIVE
          trigg_dir = ncNEGATIVE
          ref_pulse = ncOFF
          fix_dir = ncOFF
          tr_s_block = 0.0
          torque_lim = 0.0
          ds_block = 0.0
          ds_stop = 0.0
      basis:
        parameter:
          v_pos = 4000.0
          v_neg = 4000.0
          a1_pos = 10000.0
          a2_pos = 10000.0
          a1_neg = 10000.0
          a2_neg = 10000.0
    message:
      text:
        parameter:
          format = ncBREAK
          columns = 80
          data_modul
```

### Data object Logical/acp10etxen (Ett)

- acp10etxen.ett (not shown)

### Package Logical/gAxis03obj - gAxis03obj

- Data object Logical/gAxis03obj/gAxis03a (Apt) (no source held here)

### Data object Logical/gAxis03obj/gAxis03i (Ax)

#### gAxis03i.ax
```
InitParameter (Version=3.13.1, NcSwId=Acp10)
  ACP10AXIS_typ:
    dig_in:
      level:
        reference = ncACTIV_HI
        pos_hw_end = ncACTIV_HI
        neg_hw_end = ncACTIV_HI
        trigger1 = ncACTIV_HI
        trigger2 = ncACTIV_HI
    encoder_if:
      parameter:
        count_dir = ncSTANDARD
        scaling:
          load:
            units = 1000
            rev_motor = 1
    limit:
      parameter:
        v_pos = 7500.0
        v_neg = 7500.0
        a1_pos = 10000.0
        a2_pos = 10000.0
        a1_neg = 10000.0
        a2_neg = 10000.0
        t_jolt = 0
        t_in_pos = 0
        pos_sw_end = 8388607
        neg_sw_end = -8388607
        ds_warning = 500
        ds_stop = 50000.0
        a_stop = 1.0E+30
        dv_stop = 0
        dv_stop_mode = ncOFF
    controller:
      mode = ncPOSITION
      position:
        kv = 10.0
        tn = 0
        t_predict = 0.04
        t_total = 0.04
        p_max = 10000.0
        i_max = 0
      speed:
        kv = 2.0
        tn = 0
        t_filter = 0.0
        isq_filter1:
          type = ncOFF
          a0 = 0.0
          a1 = 0.0
          b0 = 0.0
          b1 = 0.0
          b2 = 0.0
          c0_par_id = 0
          c1_par_id = 0
        isq_filter2:
          type = ncOFF
          a0 = 0.0
          a1 = 0.0
          b0 = 0.0
          b1 = 0.0
          b2 = 0.0
          c0_par_id = 0
          c1_par_id = 0
        isq_filter3:
          type = ncOFF
          a0 = 0.0
          a1 = 0.0
          b0 = 0.0
          b1 = 0.0
          b2 = 0.0
          c0_par_id = 0
          c1_par_id = 0
      uf:
        type = ncLINEAR
        auto_config = ncMOTOR_PAR
        u0 = 0
        un = 0
        fn = 50.0
        k_f_slip = 0
      ff:
        torque_load = 0.0
        torque_pos = 0.0
        torque_neg = 0.0
        kv_torque = 0.0
        inertia = 0.0
        t_filter_a = 0.0
    move:
      stop:
        parameter[0]:
          decel_ramp = ncA_LIMIT
          controller = ncON
        parameter[1]:
          decel_ramp = ncA_LIMIT
          controller = ncON
        parameter[2]:
          decel_ramp = ncA_LIMIT
          controller = ncON
        parameter[3]:
          decel_ramp = ncA_LIMIT
          controller = ncON
        quickstop:
          decel_ramp = ncA_LIMIT
        drive_error:
          decel_ramp = ncA_LIMIT
      homing:
        parameter:
          s = 0
          v_switch = 6000.0
          v_trigger = 2000.0
          a = 10000.0
          mode = ncEND_SWITCH
          edge_sw = ncNEGATIVE
          start_dir = ncPOSITIVE
          trigg_dir = ncNEGATIVE
          ref_pulse = ncOFF
          fix_dir = ncOFF
          tr_s_block = 0
          torque_lim = 0
          ds_block = 0
          ds_stop = 0
      basis:
        parameter:
          v_pos = 4000.0
          v_neg = 4000.0
          a1_pos = 10000.0
          a2_pos = 10000.0
          a1_neg = 10000.0
          a2_neg = 10000.0
    message:
      text:
        parameter:
          format = ncBREAK
          columns = 80
          data_modul = acp10etxen
```

### Program Logical/SDCAxisCtrl_X (ANSIC)

#### Main.c - Init, cyclic, exit code
```c
#include <bur/plctypes.h>

#ifdef _DEFAULT_INCLUDES
	#include <AsDefault.h>
#endif

void increase_counters(void);
void Homing(void);

void _INIT ProgramInit(void)
{
	//Устанваливаем типы SDC модулей
	AxisX_HW.EncIf1_Typ = ncSDC_ENC16;
	AxisX_HW.DiDoIf_Typ = ncSDC_DIDO;
	AxisX_HW.DrvIf_Typ = ncSDC_DRVSERVO16;

	//Устанавливаем имена переменных
	strcpy(AxisX_HW.EncIf1_Name, "AxisX_EncIf");
	strcpy(AxisX_HW.DrvIf_Name, "AxisX_DrvIf");
	strcpy(AxisX_HW.DiDoIf_Name, "AxisX_DiDoIf");

	//Устанавливаем входы готовности и нормальной работы
	AxisX_EncIf.iEncOK = 1;
	AxisX_DrvIf.iDrvOK = 1;
	AxisX_DrvIf.iStatusEnable = 1;
	AxisX_DiDoIf.iDriveReady = 1;

	fb_regulator.dt = 0.002;
	fb_regulator.k_i = 0.16;
	fb_regulator.k_p = 0.0064;
	fb_regulator.max_abc_value = 24.0;

	pwm_period = 200;
}

void _CYCLIC ProgramCyclic(void)
{
	increase_counters();
	AxisX_EncIf.iActTime = (INT)AsIOTimeCyclicStart();
	AxisX_DiDoIf.iPosHwEnd = axis_X.endswitch_a_reached;
	AxisX_DiDoIf.iNegHwEnd = axis_X.endswitch_b_reached;

	if(coil_powered_X == 1)
	{
		/*if(!Already_Homed)
		{
			Homing();
		}
		else
		{*/
			increase_counters();
			axis_X.reset_counter = 0;
			FB_Axis(&axis_X);
			coil_pwm_value = 32767;
		AxisX_DiDoIf.iPosHwEnd = axis_X.endswitch_a_reached;
		AxisX_DiDoIf.iNegHwEnd = axis_X.endswitch_b_reached;
			FB_Axis(&axis_X);

			fb_regulator.e = (AxisX_DrvIf.oSetPos*100)  - axis_X.speed;//oSetPos;
			FB_Regulator(&fb_regulator);

			axis_X.u = fb_regulator.u ;
			FB_Axis(&axis_X);//}
	}
	else
	{
		coil_pwm_value = 0;
		fb_regulator.e = 0 ;
		FB_Regulator(&fb_regulator);
		axis_X.u = 0;
		FB_Axis(&axis_X);

	}
	// COUNTER1 = axis_X.counter

	//COUNTER2 += axis_X.counter - COUNTER1;
}

void increase_counters(void)
{
	AxisX_EncIf.iLifeCnt++;
	AxisX_DiDoIf.iLifeCntDriveEnable++;
	AxisX_DiDoIf.iLifeCntDriveReady++;
	AxisX_DiDoIf.iLifeCntNegHwEnd++;
	AxisX_DiDoIf.iLifeCntPosHwEnd++;
	AxisX_DiDoIf.iLifeCntReference++;
	AxisX_DrvIf.iLifeCnt++;
}

void Homing(void)
{
	increase_counters();
	coil_pwm_value = 32767;
	iPosHwEnd = axis_X.endswitch_a_reached;
	iNegHwEnd = axis_X.endswitch_b_reached;
	FB_Axis(&axis_X);

	fb_regulator.e = (AxisX_DrvIf.oSetPos * 10) - axis_X.speed;//oSetPos;
	FB_Regulator(&fb_regulator);

	axis_X.u = fb_regulator.u ;
	FB_Axis(&axis_X);
	if (iPosHwEnd)
	{
		coil_pwm_value = 0;
		fb_regulator.e = 0;
		FB_Regulator(&fb_regulator);
		axis_X.u = 0;
		FB_Axis(&axis_X);
		axis_X.reset_counter = 1;
		FB_Axis(&axis_X);
		if(k == 200)
		{
			Already_Homed = 1;
			FB_Axis(&axis_X);
		}
		k++;

	}

}

void _EXIT ProgramExit(void)
{
	// Insert code here

}
```

#### Variables.var - Local variables
```iecst
VAR
	min_task : INT := 7000;
	desired_speed : INT := 0;
	axis_X : FB_Axis;
	coil_powered_X : BOOL := FALSE;
	coil_pwm_value : {REDUND_UNREPLICABLE} INT := 200;
	fb_controller : FB_Controller;
	pwm_period : {REDUND_UNREPLICABLE} UINT := 200;
	Already_Homed : BOOL := FALSE;
	k : INT := 0;
	reset : BOOL := FALSE;
END_VAR
```

### Program Logical/ncsdcctrl (IEC)

#### ncsdcctrl.var
```iecst
VAR
	gAxis05_oSetPosOld : INT := 0;
END_VAR
```

#### ncsdcctrlCyclic.st
```iecst
PROGRAM _CYCLIC

(* ### BEGIN gAxis05 ### *)

(* life counter emulation of digital inputs *)
      gAxis05_DiDoIf.iLifeCntReference := gAxis05_DiDoIf.iLifeCntReference + 1;
      gAxis05_DiDoIf.iLifeCntNegHwEnd  := gAxis05_DiDoIf.iLifeCntNegHwEnd  + 1;
      gAxis05_DiDoIf.iLifeCntPosHwEnd  := gAxis05_DiDoIf.iLifeCntPosHwEnd  + 1;

(* default function model of ACOPOSmicro: convert absolute steps to delta steps - overflow save delta calculation *)
      gAxis05_MotorStep0 := gAxis05_DrvIf.oSetPos - gAxis05_oSetPosOld;
      gAxis05_oSetPosOld := gAxis05_DrvIf.oSetPos;

(* ### END gAxis05 ### *)

END_PROGRAM
```

#### ncsdcctrlInit.st
```iecst
PROGRAM _INIT

(* ### BEGIN gAxis05 ### *)

(* initialize general interfaces *)
      gAxis05.size := gAxis05.size;
      gAxis05_HW.DrvIf_Typ := ncSDC_DRVSM16;
      brsstrcpy( ADR(gAxis05_HW.DrvIf_Name[0]), ADR('gAxis05_DrvIf') );
      gAxis05_HW.DiDoIf_Typ := ncSDC_DIDO;
      brsstrcpy( ADR(gAxis05_HW.DiDoIf_Name[0]), ADR('gAxis05_DiDoIf') );
      gAxis05_HW.EncIf1_Typ := ncSDC_ENC16;
      brsstrcpy( ADR(gAxis05_HW.EncIf1_Name[0]), ADR('gAxis05_EncIf1') );
      gAxis05_EncIf1.iLifeCnt := gAxis05_EncIf1.iLifeCnt;

(* initialize old-value for delta step calculation *)
      gAxis05_oSetPosOld := gAxis05_DrvIf.oSetPos;

(* ### END gAxis05 ### *)

END_PROGRAM
```

### Package Logical/gAxis05obj - gAxis05obj

### Data object Logical/gAxis05obj/gAxis05a (Apt)

#### gAxis05a.apt
```
AcoposParameterTable:
  Root Parameters:
    64232 = 51200 (Name=SM_SCALE_STEP)
    64233 = 1000 (Name=SM_SCALE_LOAD_UNITS)
    64234 = 1 (Name=SM_SCALE_LOAD_MOTREV)
    109 = 1024 (Name=SCALE_ENCOD_INCR)
```

- Data object Logical/gAxis05obj/gAxis05i (Ax) (no source held here)

### Program Logical/SDCAxisCtrl_Y (ANSIC)

#### Variables.var
```iecst
VAR
	min_task : INT := 7000;
	desired_speed : INT := 0;
	gaxis03 : FB_Axis;
	coil_powered_Y : BOOL := FALSE;
	coil_pwm_value : {REDUND_UNREPLICABLE} INT := 200;
	fb_controller : FB_Controller;
	pwm_period : {REDUND_UNREPLICABLE} UINT := 200;
	Already_Homed : BOOL := FALSE;
	k : INT := 0;
	reset : BOOL := FALSE;
END_VAR
```

#### Main.c
```c
#include <bur/plctypes.h>

#ifdef _DEFAULT_INCLUDES
#include <AsDefault.h>
#endif

void increase_counters(void);
void Homing(void);

void _INIT ProgramInit(void)
{
	//Устанваливаем типы SDC модулей
	gAxis03_HW.EncIf1_Typ = ncSDC_ENC16;
	gAxis03_HW.DiDoIf_Typ = ncSDC_DIDO;
	gAxis03_HW.DrvIf_Typ = ncSDC_DRVSERVO16;

	//Устанавливаем имена переменных
	strcpy(gAxis03_HW.EncIf1_Name, "gAxis03_EncIf");
	strcpy(gAxis03_HW.DrvIf_Name, "gAxis03_DrvIf");
	strcpy(gAxis03_HW.DiDoIf_Name, "gAxis03_DiDoIf");

	//Устанавливаем входы готовности и нормальной работы
	gAxis03_EncIf.iEncOK = 1;
	gAxis03_DrvIf.iDrvOK = 1;
	gAxis03_DrvIf.iStatusEnable = 1;
	gAxis03_DiDoIf.iDriveReady = 1;

	fb_regulator.dt = 0.002;
	fb_regulator.k_i = 0.16;
	fb_regulator.k_p = 0.0064;
	fb_regulator.max_abc_value = 24.0;

	pwm_period = 200;
}

void _CYCLIC ProgramCyclic(void)
{
	increase_counters();
	gAxis03_EncIf.iActTime = (INT)AsIOTimeCyclicStart();
	gAxis03_DiDoIf.iPosHwEnd = gaxis03.endswitch_a_reached;
	gAxis03_DiDoIf.iNegHwEnd = gaxis03.endswitch_b_reached;

	if(coil_powered_Y == 1)
	{
		/*if(!Already_Homed)
		{
			Homing();
		}
		else
		{*/
		increase_counters();
		gaxis03.reset_counter = 0;
		FB_Axis(&gaxis03);
		coil_pwm_value = 32767;
		gAxis03_DiDoIf.iPosHwEnd = gaxis03.endswitch_a_reached;
		gAxis03_DiDoIf.iNegHwEnd = gaxis03.endswitch_b_reached;
		FB_Axis(&gaxis03);

		fb_regulator.e = (gAxis03_DrvIf.oSetPos*100)  - gaxis03.speed;//oSetPos;
		FB_Regulator(&fb_regulator);

		gaxis03.u = fb_regulator.u ;
		FB_Axis(&gaxis03);//}
	}
	else
	{
		coil_pwm_value = 0;
		fb_regulator.e = 0 ;
		FB_Regulator(&fb_regulator);
		gaxis03.u = 0;
		FB_Axis(&gaxis03);

	}
	// COUNTER1 = axis_X.counter

	//COUNTER2 += axis_X.counter - COUNTER1;
}

void increase_counters(void)
{
	gAxis03_EncIf.iLifeCnt++;
	gAxis03_DiDoIf.iLifeCntDriveEnable++;
	gAxis03_DiDoIf.iLifeCntDriveReady++;
	gAxis03_DiDoIf.iLifeCntNegHwEnd++;
	gAxis03_DiDoIf.iLifeCntPosHwEnd++;
	gAxis03_DiDoIf.iLifeCntReference++;
	gAxis03_DrvIf.iLifeCnt++;
}

void Homing(void)
{/*
	increase_counters();
	coil_pwm_value = 32767;
	iPosHwEnd = axis_X.endswitch_a_reached;
	iNegHwEnd = axis_X.endswitch_b_reached;
	FB_Axis(&axis_X);

	fb_regulator.e = (AxisX_DrvIf.oSetPos * 10) - axis_X.speed;//oSetPos;
	FB_Regulator(&fb_regulator);

	axis_X.u = fb_regulator.u ;
	FB_Axis(&axis_X);
	if (iPosHwEnd)
	{
		coil_pwm_value = 0;
		fb_regulator.e = 0;
		FB_Regulator(&fb_regulator);
		axis_X.u = 0;
		FB_Axis(&axis_X);
		axis_X.reset_counter = 1;
		FB_Axis(&axis_X);
		if(k == 200)
		{
			Already_Homed = 1;
			FB_Axis(&axis_X);
		}
		k++;

	}
	*/
}

void _EXIT ProgramExit(void)
{
	// Insert code here

}
```

### Program Logical/SDCAxisCtrl_Z (ANSIC)

#### Variables.var
```iecst
VAR
	min_task : INT := 7000;
	desired_speed : INT := 0;
	gaxis05 : FB_Axis;
	coil_powered_Z : BOOL := FALSE;
	coil_pwm_value : {REDUND_UNREPLICABLE} INT := 200;
	fb_controller : FB_Controller;
	pwm_period : {REDUND_UNREPLICABLE} UINT := 200;
	Already_Homed : BOOL := FALSE;
	k : INT := 0;
	reset : BOOL := FALSE;
END_VAR
```

#### Main.c
```c
#include <bur/plctypes.h>

#ifdef _DEFAULT_INCLUDES
#include <AsDefault.h>
#endif

void increase_counters(void);
void Homing(void);

void _INIT ProgramInit(void)
{
	//Устанваливаем типы SDC модулей
	gAxis05_HW.EncIf1_Typ = ncSDC_ENC16;
	gAxis05_HW.DiDoIf_Typ = ncSDC_DIDO;
	gAxis05_HW.DrvIf_Typ = ncSDC_DRVSERVO16;

	//Устанавливаем имена переменных
	strcpy(gAxis05_HW.EncIf1_Name, "gAxis05_EncIf");
	strcpy(gAxis05_HW.DrvIf_Name, "gAxis05_DrvIf");
	strcpy(gAxis05_HW.DiDoIf_Name, "gAxis05_DiDoIf");

	//Устанавливаем входы готовности и нормальной работы
	gAxis05_EncIf.iEncOK = 1;
	gAxis05_DrvIf.iDrvOK = 1;
	gAxis05_DrvIf.iStatusEnable = 1;
	gAxis05_DiDoIf.iDriveReady = 1;

	fb_regulator.dt = 0.002;
	fb_regulator.k_i = 0.16;
	fb_regulator.k_p = 0.0064;
	fb_regulator.max_abc_value = 24.0;

	pwm_period = 200;
}

void _CYCLIC ProgramCyclic(void)
{
	increase_counters();
	gAxis05_EncIf.iActTime = (INT)AsIOTimeCyclicStart();
	gAxis05_DiDoIf.iPosHwEnd = gaxis05.endswitch_a_reached;
	gAxis05_DiDoIf.iNegHwEnd = gaxis05.endswitch_b_reached;

	if(coil_powered_Z == 1)
	{
		/*if(!Already_Homed)
		{
			Homing();
		}
		else
		{*/
		increase_counters();
		gaxis05.reset_counter = 0;
		FB_Axis(&gaxis05);
		coil_pwm_value = 32767;
		gAxis05_DiDoIf.iPosHwEnd = gaxis05.endswitch_a_reached;
		gAxis05_DiDoIf.iNegHwEnd = gaxis05.endswitch_b_reached;
		FB_Axis(&gaxis05);

		fb_regulator.e = (gAxis05_DrvIf.oSetPos*100)  - gaxis05.speed;//oSetPos;
		FB_Regulator(&fb_regulator);

		gaxis05.u = fb_regulator.u ;
		FB_Axis(&gaxis05);//}
	}
	else
	{
		coil_pwm_value = 0;
		fb_regulator.e = 0 ;
		FB_Regulator(&fb_regulator);
		gaxis05.u = 0;
		FB_Axis(&gaxis05);

	}
	// COUNTER1 = axis_X.counter

	//COUNTER2 += axis_X.counter - COUNTER1;
}

void increase_counters(void)
{
	gAxis05_EncIf.iLifeCnt++;
	gAxis05_DiDoIf.iLifeCntDriveEnable++;
	gAxis05_DiDoIf.iLifeCntDriveReady++;
	gAxis05_DiDoIf.iLifeCntNegHwEnd++;
	gAxis05_DiDoIf.iLifeCntPosHwEnd++;
	gAxis05_DiDoIf.iLifeCntReference++;
	gAxis05_DrvIf.iLifeCnt++;
}

void Homing(void)
{/*
	increase_counters();
	coil_pwm_value = 32767;
	iPosHwEnd = axis_X.endswitch_a_reached;
	iNegHwEnd = axis_X.endswitch_b_reached;
	FB_Axis(&axis_X);

	fb_regulator.e = (AxisX_DrvIf.oSetPos * 10) - axis_X.speed;//oSetPos;
	FB_Regulator(&fb_regulator);

	axis_X.u = fb_regulator.u ;
	FB_Axis(&axis_X);
	if (iPosHwEnd)
	{
		coil_pwm_value = 0;
		fb_regulator.e = 0;
		FB_Regulator(&fb_regulator);
		axis_X.u = 0;
		FB_Axis(&axis_X);
		axis_X.reset_counter = 1;
		FB_Axis(&axis_X);
		if(k == 200)
		{
			Already_Homed = 1;
			FB_Axis(&axis_X);
		}
		k++;

	}
	*/
}

void _EXIT ProgramExit(void)
{
	// Insert code here

}
```

### Data object Logical/CncInit (Cns)

- CncInit.cns - ARNC0 init object for CNC (not shown)

### Data object Logical/CncProg (Cnc)

#### CncProg.cnc - CNC program (G-Code)
```
%001 (CncProgram)

( TODO: Add code here )

N10 G90
N20 F390000
N30 G01 X0 Y65913 Z0
N40 G01 X0 Y65913 Z65913
N50 G01 X65913 Y0 Z65913
N60 G01 X0 Y0 Z65913
N70 G01 X0 Y0 Z0
N999 M30
```

### Data object Logical/GmcIpConfig/gmcipsys (Cnc, version 5.02.1)

#### gmcipsys.cnc
```
LANGS (defaultLangId=1, defaultDataLangId=3)
  CMDQUEUE (BufferSize=15)
  MEM (ReserveMB=5, LimitPercent=80%)
  EXEC (InstrBurstBG=200, CycleBurstBG=0, Stack=16384, MinorStack=2048, EStack=1024)
  LOAD (ReadLineBurstMax=100, ReadLineBurstMin=20, ParseLineBurstMax=10, ParseLineBurstMin=2, RuntimeIOBlocking=No)
  DISABLE_MSG = 15238 
    15336 
    15337 
    15666 
    15784 
    15864 
    15740
  LANG (langId=1, langName=B&R GCode, langModule=ailgcode)
    LANGCONFIG gmciplbr
    LANGCONFIG gmcipcbr
    LANGCONFIG gmcipubr
    FILEEXT .cnc
    FILEEXT .prg
    MAINSEARCHPATH $ (FileDevice=CNC_PrgDir)
    MAINSEARCHPATH $ (DataObject=Yes)
    INCLUDEPATH $ (FileDevice=CNC_PrgDir)
    INCLUDEPATH $ (DataObject=Yes)
  LANG (langId=2, langName=Alternative Language 1 GCode, langModule=ailgcode)
    LANGCONFIG gmciplsm
    LANGCONFIG gmcipcbr
    LANGCONFIG gmcipcsm
    LANGCONFIG gmcipusm
    FILEPREFIX = _N_
    FILEEXT = .MPF
    FILEEXT = _MPF
    FILEEXT = .SPF
    FILEEXT = _SPF
    MAINSEARCHPATH = \$ (FileDevice=CNC_PrgDir)
    MAINSEARCHPATH = \_N_MPF_DIR\$ (FileDevice=CNC_PrgDir)
    MAINSEARCHPATH = \_N_SPF_DIR\$ (FileDevice=CNC_PrgDir)
    MAINSEARCHPATH = $ (DataObject=1)
    INCLUDEPATH = \$ (FileDevice=CNC_PrgDir)
    INCLUDEPATH = \_N_SPF_DIR\$ (FileDevice=CNC_PrgDir)
    INCLUDEPATH = \_N_MPF_DIR\$ (FileDevice=CNC_PrgDir)
    INCLUDEPATH = $ (DataObject=1)
  LANG (langId=3, langName=IEC-ST, langModule=ailgcode)
    LANGCONFIG gmcipiec
    LANGCONFIG gmcipmx (RequireFnIgnore=MXConvertOrient)
    LANGCONFIG gmcipui (IfNotExist=Warn)
    FILEEXT .typ (DeclScope=IP_GLOBAL)
    FILEEXT .var (DeclScope=IP_GLOBAL)
    FILEEXT .fun (DeclScope=IP_GLOBAL)
    FILEEXT .iec (DeclScope=IP_LOCAL)
    FILEEXT .st (DeclScope=IP_LOCAL)
    FILEEXT _iec (DeclScope=IP_LOCAL)
    MAINSEARCHPATH = \$ (FileDevice=IEC_PrgDir)
    MAINSEARCHPATH = \$ (FileDevice=CNC_PrgDir)
    MAINSEARCHPATH \TYP\$ (FileDevice=CNC_PrgDir, DataObject=No)
    INCLUDEPATH = \$ (FileDevice=IEC_PrgDir)
    INCLUDEPATH = \$ (FileDevice=CNC_PrgDir)
    INCLUDEPATH \TYP\$ (FileDevice=CNC_PrgDir, DataObject=No)
  XML_INCLUDE gmcipus (IfNotExist=Warn)
```

### Data object Logical/GmcIpConfig/gmciplbr (Cnc, version 5.02.1)

#### gmciplbr.cnc
```
Root (LangModule=ailgcode, Version=1.0)
  BuiltInProcs:
    cancel = beginpathsynch
        StopCyclicGroups(:${*}:);
      endpathsynch (MinArgs=1, MaxArgs=*)
  BuiltInFns (PatternSuffix=:\[)
    ABS = Abs(:$[1]:) (NumArgs=1, Inline=Yes)
    SQR = ($[1] * $[1]) (NumArgs=1)
    ACOS = ACos(:$[1]:) (NumArgs=1, Inline=Yes)
    ASIN = ASin(:$[1]:) (NumArgs=1, Inline=Yes)
    ATAN = ATan(:$[1]:) (NumArgs=1, Inline=Yes)
    COS = Cos(:$[1]:) (NumArgs=1, Inline=Yes)
    DEXP = DExp(:$[1]:) (NumArgs=1, Inline=Yes)
    EXP = Exp(:$[1]:) (NumArgs=1, Inline=Yes)
    FIX = Fix(:$[1]:) (NumArgs=1, Inline=Yes)
    FRACT = Fract(:$[1]:) (NumArgs=1, Inline=Yes)
    FUP = Fup(:$[1]:) (NumArgs=1, Inline=Yes)
    INV = ~($[1]) (NumArgs=1, Inline=Yes)
    LN = Ln(:$[1]:) (NumArgs=1, Inline=Yes)
    LOG = Log(:$[1]:) (NumArgs=1, Inline=Yes)
    ROUND = ToInt(:$[1]:) (NumArgs=1, Inline=Yes)
    SIN = Sin(:$[1]:) (NumArgs=1, Inline=Yes)
    SQRT = Sqrt(:$[1]:) (NumArgs=1, Inline=Yes)
    TAN = Tan(:$[1]:) (NumArgs=1, Inline=Yes)
    BOOL = ToBool(:$[1]:) (NumArgs=1, Inline=Yes)
    INT = Fix(:$[1]:) (NumArgs=1, Inline=Yes)
    ADR = Adr(:\$[1]:) (NumArgs=1, Inline=Yes)
    SIZEOF = Sizeof(:\$[1]:) (NumArgs=1, Inline=Yes)
    NUM_LOADED_FILES = NumLoadedFiles(::) (NumArgs=0)
    NUM_LOADED_PROG_FILES = NumLoadedProgFiles(::) (NumArgs=0)
    MEM_SIZE_IP_ALL = MemSizeIpInstAll(::) (NumArgs=0)
    MEM_SIZE_IP_LIB = MemSizeIpInst(::) (NumArgs=0)
    MEM_SIZE_SHLIB = MemSizeShLib(::) (NumArgs=0)
    MEM_SIZE_FILE = MemSizeFile(:$[1]:) (MinArgs=0, MaxArgs=1)
    MEM_SIZE_IP_STACK_SPACE = MemStackSpace(::) (NumArgs=0)
  AxesSpec:
    AxisRef = $\s*=\s*AC (Mode=3)
    AxisRef = $\s*=\s*IC (Mode=4)
  PVMacros:
    RDISABLE (ArrayDims=0, Group=500)
      CALL = @#job->sa.keep_alive = 1;
        @#thread.sa_keep_alive = 1; (Inline=Yes)
  Parameters:
    R (IndexType=RParamIndex, ValueType=FLOAT)
      ARG (ref=EXPR, DataType=RParamIndex)
    P (IndexType=RParamIndex, ValueType=FLOAT)
      ARG (ref=EXPR, DataType=RParamIndex)
    EXB (IndexType=EXParamIndex, ValueType=Byte)
      ARG (ref=EXPR, DataType=EXParamIndex)
    EXW (IndexType=EXParamIndex, ValueType=Word)
      ARG (ref=EXPR, DataType=EXParamIndex)
    EXL (IndexType=EXParamIndex, ValueType=Long)
      ARG (ref=EXPR, DataType=EXParamIndex)
    EXF (IndexType=EXFParamIndex, ValueType=FLOAT)
      ARG (ref=EXPR, DataType=EXFParamIndex)
    MW (Synchronous=Yes, IndexType=MParamIndex, ValueType=Word)
      ARG (ref=EXPR, DataType=MParamIndex)
    ML (Synchronous=Yes, IndexType=MParamIndex, ValueType=Long)
      ARG (ref=EXPR, DataType=MParamIndex)
    MF (Synchronous=Yes, IndexType=MParamIndex, ValueType=FLOAT)
      ARG (ref=EXPR, DataType=MParamIndex)
  PrimTypes (PatternSuffix=:[^\[], MapIECTypes=Yes)
  Preprocess:
    PP_RULE_FRAME_I (Search=$FRAME_I, Replace=[1,0,0,0,1,0,0,0,1,0,0,0])
    PP_RULE_FRAME_DEF (IsPattern=Yes, Search=FRAME:[^\w\d], Replace=LREAL{12})
  FubTemplates:
    StdFubTemplate (IsDefault=Yes, Inline=Yes)
      Arg (ref=FUBINST, DataType=FLOAT)
      Arg (ref=FUBERRLEV, DataType=FLOAT)
      Arg (ref=PATHSYNCH, DataType=FLOAT)
      Arg (ref=BLOCKING, DataType=FLOAT)
  SynchActions:
    SABlocks:
      default (IsDefault=Yes)
        cyclic (Inline=Yes)
          Arg (ref=ACTIONS, DataType=STATEMENTS)
          Arg (ref=ID, DataType=FLOAT, DefaultInt=-1, MinCount=0, MaxCount=1)
      whenever:
        cyclic (Inline=Yes)
          Arg (ref=COND, DataType=FLOAT)
          Arg (ref=ACTIONS, DataType=STATEMENTS)
          Arg (ref=ID, DataType=FLOAT, DefaultInt=-1, MinCount=0, MaxCount=1)
      when:
        cyclic (Inline=Yes)
          Arg (ref=COND, DataType=FLOAT)
          Arg (ref=ACTIONS, DataType=STATEMENTS)
          Arg (ref=ID, DataType=FLOAT, DefaultInt=-1, MinCount=0, MaxCount=1)
      every:
        cyclic (Inline=Yes)
          Arg (ref=COND, DataType=FLOAT)
          Arg (ref=ACTIONS, DataType=STATEMENTS)
          Arg (ref=ID, DataType=FLOAT, DefaultInt=-1, MinCount=0, MaxCount=1)
      from:
        cyclic (Inline=Yes)
          Arg (ref=COND, DataType=FLOAT)
          Arg (ref=ACTIONS, DataType=STATEMENTS)
          Arg (ref=ID, DataType=FLOAT, DefaultInt=-1, MinCount=0, MaxCount=1)
    NonModalActivation:
      Start = @#thread.sa_last_keep_alive = 1;
        ActivateCyclicGroup(:-1:);
      Stop = WaitStopCyclicGroups(:(:-1:):);
  ParserData (NestedComments=Yes, DefaultCaseSensitive=No, CommentsSpanLines=No, SubDeclsLocalToFile=Yes, ProgDeclsLocalToFile=Yes, AllowUnprefixedFileCalls=No, LocalVarScopeForMainProg=No, FileScopeVarsVisibleInSub=Yes, MainPrgReturnAtNextMainPrgHdr=Yes, MaxSizePassByValue=1024, AllowVarReadBeforeAssign=No, AllowArrayRefWithoutIndex=Yes, AllowStructMemberAutoDereference=Yes, AllowVariableAutoDereference=Yes, AllowIgnoredExtraSubArgs=Yes, EnableStringCharacterIndexing=Yes, OnMacroRedefinition=Warn, CheckFileTimestampBeforeCalls=Yes)
    TKG_END_OF_LINE = \n (IsPattern=No)
    TKG_LINE_CONTINUE = \ (IsPattern=No, FileXLInvalid=Yes)
    TKG_LINE_BREAK = @@
    TKG_ARITH_BINARY_MODULO = MOD
    TKG_TRUE = TRUE:\W (IsPattern=Yes)
    TKG_FALSE = FALSE:\W (IsPattern=Yes)
    TKG_PAREVAL_MODAL_ID = ID:[\s=] (FileXLInvalid=Yes, IsPattern=Yes)
    TKG_OPEN_COMMENT = (
    TKG_CLOSE_COMMENT = )
    TKG_OPEN_BRACKET = [
    TKG_COMMA = ,
    TKG_CLOSE_BRACKET = ]
    TKG_OPEN_INDEXBRACKET = {
    TKG_CLOSE_INDEXBRACKET = }
    TKG_NUMBER = \d+\.\d+|\d+\.:[^\.] (IsPattern=Yes)
    TKG_INTEGER = \d+ (IsPattern=Yes)
    TKG_FRACTION = \.\d+ (IsPattern=Yes)
    TKG_DOT = \.:\w (IsPattern=Yes, FollowedBy=TKG_STRUCT_MEMBER_REF)
    TKG_STRUCT_MEMBER_REF = \w|\w[\w\d]+ (IsPattern=Yes, Restricted=Yes)
    TKG_NUMBER_EXP = EX:[\s\d\+\-\.] (IsPattern=Yes)
    TKG_MACRO_DEFINE_GLOBAL = define\s+ip_global:\s (IsPattern=Yes, FollowedBy=TKG_MACRO_NAME)
    TKG_MACRO_DEFINE = define\s+local:\s|define:\s (IsPattern=Yes, FollowedBy=TKG_MACRO_NAME)
    TKG_MACRO_UNDEFINE = undefine:\s (IsPattern=Yes, FollowedBy=TKG_MACRO_NAME)
    TKG_MACRO_AS = as:[\s\n] (IsPattern=Yes, FollowedBy=TKG_MACRO_TEXT)
    TKG_MACRO_NAME = [$\w][$\w\d]+ (Restricted=Yes, IsPattern=Yes)
    TKG_MACRO_TEXT = . (Restricted=Yes, IsPattern=Yes)
    TKG_BUILTIN_NUM_FN_NAME
    _TKG_LABEL_DEF1:
      TKG_LABEL_DEF = L[\w\d]+:\:[^\w\d] (IsPattern=Yes, FollowedBy=TKG_LABEL_SUFFIX)
    TKG_SUBPROG_START = %:L (FileXLInvalid=Yes, IsPattern=Yes, FollowedBy=TKG_SUBPROG_NAME)
    TKG_SUBPROG_NAME = L\d+ (IsPattern=Yes, Restricted=Yes)
    TKG_SUBPROG_CALL = L:L\d (IsPattern=Yes, FollowedBy=TKG_SUBPROG_NAME)
    TKG_SUBPROG_PROTO = %D:L (IsPattern=Yes, FollowedBy=TKG_SUBPROG_NAME)
    TKG_SUBCALL_REPEAT_PREFIX = O:[\s\d] (IsPattern=Yes, FollowedBy=TKG_INTEGER)
    TKG_EXTERN = EXTERN:\s (IsPattern=Yes, FollowedBy=TKG_PROG_FILE_NAME)
    TKG_ARG_PASSBYREF = VAR\s (IsPattern=Yes)
    TKG_SET_MODAL_SUB = MCALL:\W (FileXLInvalid=Yes, IsPattern=Yes)
    TKG_PROG_START = %:\d (IsPattern=Yes, FollowedBy=TKG_PROG_NAME)
    TKG_PROG_NAME = \d+ (IsPattern=Yes, Restricted=Yes)
    TKG_PROG_CALL = L:[^L] (IsPattern=Yes, FollowedBy=TKG_PROG_FILE_NAME)
    TKG_PROG_FILE_NAME = [\^#&@']?[\w\d\.\\]+:[^\w\d\.\\\:]|[\^#][\w\d]+\:[\w\d\.\\]+ (IsPattern=Yes, Restricted=Yes)
    TKG_SUPPRESS_SINGLE_STEP = NOHALT
    TKG_NC_BLOCK_PREFIX = N:[\d\s] (IsPattern=Yes)
    TKG_PARAM_PREFIX = R:\d|P:\d|M[WLF]:\d|EX[WLBF]:\d (IsPattern=Yes)
    TKG_SUBRANGE = ..
    TKG_G_CODE_PREFIX = G:[\s\d] (IsPattern=Yes)
    TKG_M_CODE_PREFIX = M:[\s\d\[] (IsPattern=Yes)
    TKG_PAREVAL_DO = do:\s (FileXLInvalid=Yes, IsPattern=Yes)
    TKG_GOTO = $GOTO:\s (FileXLInvalid=Yes, IsPattern=Yes, OptFollowedBy=TKG_GOTO_DEST)
    TKG_GOTO_DEST = \w[\w\d]* (IsPattern=Yes, Restricted=Yes)
    TKG_LOGICAL_BINARY_AND = &&
    TKG_LOGICAL_BINARY_OR = ||
    TKG_LOGICAL_BINARY_XOR = XOR
    TKG_STRING_CONCAT = <<
    TKG_COMP_BINARY_GREATER_THAN_OR_EQ = >=
    TKG_COMP_BINARY_LESS_THAN_OR_EQ = <=
    TKG_COMP_BINARY_EQUAL_TO = ==
    TKG_COMP_BINARY_NOT_EQUAL_TO = !=
    TKG_COMP_BINARY_GREATER_THAN = >
    TKG_COMP_BINARY_LESS_THAN = <
    TKG_ASSIGN_EQ = =
    TKG_LOGICAL_UNARY_NOT = !
    TKG_BITWISE_BINARY_AND = &
    TKG_BITWISE_BINARY_OR = |
    TKG_BITWISE_BINARY_XOR = ^
    TKG_BITWISE_UNARY_COMPLEMENT = ~
    TKG_ARITH_BINARY_PLUS = +
    TKG_ARITH_BINARY_MINUS = -
    TKG_ARITH_BINARY_POWER = **
    TKG_ARITH_BINARY_MULTIPLY = *
    TKG_ARITH_BINARY_DIVIDE = /
    TKG_PATHSYNCH_REC_IEC = $DO_PATH_SYNCH (FileXLInvalid=Yes)
    TKG_PATHSYNCH_END = $END_PATH_SYNCH (FileXLInvalid=Yes)
    TKG_PATHSYNCH_IPEVAL = $IP_EVAL (FileXLInvalid=Yes)
    TKG_IF = $IF (FileXLInvalid=Yes)
    TKG_THEN = $THEN (FileXLInvalid=Yes)
    TKG_BLOCK_ELSEIF = $ELSEIF (FileXLInvalid=Yes)
    TKG_BLOCK_ELSE = $ELSE (FileXLInvalid=Yes)
    TKG_BLOCK_ENDIF = $ENDIF (FileXLInvalid=Yes)
    TKG_SWITCH = $SWITCH (FileXLInvalid=Yes)
    TKG_SWITCH_CASE = $CASE (FileXLInvalid=Yes)
    TKG_SWITCH_DEFAULT = $DEFAULT (FileXLInvalid=Yes)
    TKG_ENDSWITCH = $ENDSWITCH (FileXLInvalid=Yes)
    TKG_FOR = $FOR (FileXLInvalid=Yes)
    TKG_ENDFOR = $ENDFOR (FileXLInvalid=Yes)
    TKG_WHILE = $WHILE (FileXLInvalid=Yes)
    TKG_ENDWHILE = $ENDWHILE (FileXLInvalid=Yes)
    TKG_DO = $DO (FileXLInvalid=Yes)
    TKG_ENDDO = $ENDDO (FileXLInvalid=Yes)
    TKG_BREAK = $BREAK (FileXLInvalid=Yes)
    TKG_CONTINUE = $CONTINUE (FileXLInvalid=Yes)
    TKG_PRIM_TYPE (IsPattern=Yes)
    TKG_PV_DECL = def:\s (IsPattern=Yes)
    TKG_PV_UNDECL = ~def:\s (IsPattern=Yes)
    TKG_PV_DECL_REF = \w[\w\d\.\:\*]+|\w (IsPattern=Yes, Restricted=Yes)
    TKG_VARSCOPE_IP_LOCAL = local:[\s\n] (IsPattern=Yes)
    TKG_VARSCOPE_IP_GLOBAL = ip_global:[\s\n] (IsPattern=Yes)
    TKG_VARSCOPE_NC_GLOBAL = nc_global:[\s\n] (IsPattern=Yes)
    TKG_VARSCOPE_PLC_GLOBAL = plc_global:[\s\n] (IsPattern=Yes)
    TKG_VAR_RETAIN = retain:\s (IsPattern=Yes)
    TKG_VARSYNCH_IP = ip_synch:\s (IsPattern=Yes)
    TKG_VARSYNCH_PATH = path_synch:\s (IsPattern=Yes)
    TKG_LABEL_DEF = \w:\:|\w[\w\d]+:\: (IsPattern=Yes, FollowedBy=TKG_LABEL_SUFFIX)
    TKG_LABEL_SUFFIX = : (Restricted=Yes)
    TKG_FUB_DECL = fub:\s (IsPattern=Yes)
    TKG_FUB_ERR_LEV_1 = error_level_1:\s (IsPattern=Yes)
    TKG_FUB_ERR_LEV_2 = error_level_2:\s (IsPattern=Yes)
    TKG_FUB_ERR_LEV_3 = error_level_3:\s (IsPattern=Yes)
    TKG_FUB_ERR_LEV_4 = error_level_4:\s (IsPattern=Yes)
    TKG_FUB_BLOCKING = blocking:\s (IsPattern=Yes)
    TKG_FUB_NON_BLOCKING = non_blocking:\s (IsPattern=Yes)
    TKG_IEC_TYPED_VALUE = #[\w\d]+ (IsPattern=Yes)
    TKG_REFERENCE = ref:[\s\n]|reference:[\s\n] (IsPattern=Yes, FollowedBy=TKG_IEC_TO)
    TKG_IEC_TO = to:[\s\n] (IsPattern=Yes, Restricted=Yes)
    TKG_ACCESS = ACCESS:[\s\n] (IsPattern=Yes)
    TKG_WORD = \w|\w[\w\d\.]+ (IsPattern=Yes)
  StringChars (AsciiStringStart=", UTF16StringStart=W", UTF16StringEnd=")
    EscapeSeq (Search=$N, ReplaceValue=10)
    EscapeSeq (Search=$L, ReplaceValue=10)
    EscapeSeq (Search=$P, ReplaceValue=12)
    EscapeSeq (Search=$R, ReplaceValue=13)
    EscapeSeq (Search=$T, ReplaceValue=9)
    EscapeSeq (Search=$Q, ReplaceStr=")
    EscapeSeq (Search=$', ReplaceStr=')
    EscapeSeq (Search=$", ReplaceStr=")
    EscapeSeq (Search=$[\dA-Fa-f]+, IsPattern=Yes, ReplaceEncodingBase=16)
    EscapeSeq (Search=$$, ReplaceStr=$)
    EscapeSeq (Search=$, ReplaceStr=)
```

### Data object Logical/GmcIpConfig/gmcipcbr (Cnc, version 5.02.1)

- gmcipcbr.cnc (not shown)

### Data object Logical/GmcIpConfig/gmciplsm (Cnc, version 5.02.1)

#### gmciplsm.cnc
```
Root (LangModule=ailgcode, Version=1.0)
  PrimTypes (CaseSensitive=No)
    REAL (BRType=LREAL)
    INT (BRType=DINT)
    CHAR (BRType=USINT)
    BOOL (BRType=BOOL)
    STRING (BRType=STRING)
    AXIS (BRType=AXIS)
    BR_LREAL (BRType=LREAL)
    BR_REAL (BRType=REAL)
    BR_UDINT (BRType=UDINT)
    BR_DINT (BRType=DINT)
    BR_UINT (BRType=UINT)
    BR_INT (BRType=INT)
    BR_USINT (BRType=USINT)
    BR_SINT (BRType=SINT)
    BR_BOOL (BRType=BOOL)
    BR_TIME (BRType=TIME)
    BR_DATE_AND_TIME (BRType=DATE_AND_TIME)
  Preprocess:
    PP_RULE_NCK (Search=NCK , Replace=nc_global )
    PP_RULE_CHAN (Search=CHAN , Replace=ip_global )
    PP_RULE_FRAME_I (Search=$FRAME_I, Replace=(1,0,0,0,1,0,0,0,1,0,0,0))
    PP_RULE_FRAME_DEF (IsPattern=Yes, Search=FRAME:[^\w\d], Replace=REAL[12])
  BuiltInProcs:
    cancel = beginpathsynch
        StopCyclicGroups(:${*}:);
      endpathsynch (MinArgs=1, MaxArgs=*)
    RET = #next_motion.Command = MPCMD_SET_M_FCT;
      #next_motion.Data.I4_value = 17;
      PushPacket(::);
      ReturnTo(:${*}:); (MinArgs=0, MaxArgs=4, Eval=Early, Inline=Yes)
  BuiltInFns:
    ABS = Abs(:$[1]:) (NumArgs=1, Inline=Yes)
    SIN = Sin(:$[1]:) (NumArgs=1, Inline=Yes)
    COS = Cos(:$[1]:) (NumArgs=1, Inline=Yes)
    TAN = Tan(:$[1]:) (NumArgs=1, Inline=Yes)
    ASIN = ASin(:$[1]:) (NumArgs=1, Inline=Yes)
    ACOS = ACos(:$[1]:) (NumArgs=1, Inline=Yes)
    ATAN = ATan(:$[1]:) (NumArgs=1, Inline=Yes)
    ATAN2 = ATan2(:$[1],$[2]:) (NumArgs=2, Inline=Yes)
    SQRT = Sqrt(:$[1]:) (NumArgs=1, Inline=Yes)
    POT = (($[1])*($[1])) (NumArgs=1, Inline=Yes)
    TRUNC = Fix(:$[1]:) (NumArgs=1, Inline=Yes)
    ROUND = Round(:$[1]:) (NumArgs=1, Inline=Yes)
    LN = Ln(:$[1]:) (NumArgs=1, Inline=Yes)
    EXP = Exp(:$[1]:) (NumArgs=1, Inline=Yes)
    MINVAL = MinVal(:$[1], $[2]:) (NumArgs=2, Inline=Yes)
    MAXVAL = MaxVal(:$[1], $[2]:) (NumArgs=2, Inline=Yes)
    BOUND = Bounds(:$[1], $[2], $[3]:) (NumArgs=3, Inline=Yes)
    TO_BOOL = ToBool(:$[1]:) (NumArgs=1, Inline=Yes)
    TO_INT = ToInt(:$[1]:) (NumArgs=1, Inline=Yes)
    TO_CHAR = ToChar(:$[1]:) (NumArgs=1, Inline=Yes)
    TO_REAL = ToLReal(:$[1]:) (NumArgs=1, Inline=Yes)
    TO_FLOAT = ToFloat(:$[1]:) (NumArgs=1, Inline=Yes)
    DEFINED = Defined(:$[1]:) (NumArgs=1, Inline=Yes)
    TIME_MS = TimeMs(::) (NumArgs=0)
    SET = ${*} (MinArgs=0, MaxArgs=*, Inline=Yes)
    REP = ArrayRep(:${*}:) (MinArgs=1, MaxArgs=2, Inline=Yes)
    ADR = Adr(:\$[1]:) (NumArgs=1, Inline=Yes)
    SIZEOF = Sizeof(:\$[1]:) (NumArgs=1, Inline=Yes)
    NUM_LOADED_FILES = NumLoadedFiles(::) (NumArgs=0)
    NUM_LOADED_PROG_FILES = NumLoadedProgFiles(::) (NumArgs=0)
    MEM_SIZE_IP_ALL = MemSizeIpInstAll(::) (NumArgs=0)
    MEM_SIZE_IP_LIB = MemSizeIpInst(::) (NumArgs=0)
    MEM_SIZE_SHLIB = MemSizeShLib(::) (NumArgs=0)
    MEM_SIZE_FILE = MemSizeFile(:$[1]:) (MinArgs=0, MaxArgs=1)
    MEM_SIZE_IP_STACK_SPACE = MemStackSpace(::) (NumArgs=0)
  AxesSpec:
    AxisRef = $\s*=\s*AC (Mode=3)
    AxisRef = $\s*=\s*IC (Mode=4)
  PVMacros:
    SBLOF (ArrayDims=0, Group=500)
      CALL = #call->forbid_stepping = 1; (Inline=Yes)
    SBLON (ArrayDims=0, Group=500)
      CALL = #call->forbid_stepping = 0; (Inline=Yes)
    DISPLOF (ArrayDims=0, Group=500)
      CALL = #call->forbid_display = 1; (Inline=Yes)
    DISPLON (ArrayDims=0, Group=500)
      CALL = #call->forbid_display = 0; (Inline=Yes)
    RDISABLE (ArrayDims=0, Group=500)
      CALL = @#job->sa.keep_alive = 1;
        @#thread.sa_keep_alive = 1; (Inline=Yes)
    P_SUBPAR $P_SUBPAR (ArrayDims=1, Group=500)
      GET = return ArgNumIsDefined(:$[1]:);
    P_STACK $P_STACK:
      GET = return UserCallDepth(::);
  FubTemplates:
    StdFubTemplate (IsDefault=Yes, Inline=Yes)
      Arg (ref=FUBINST, DataType=FLOAT)
      Arg (ref=FUBERRLEV, DataType=FLOAT)
      Arg (ref=PATHSYNCH, DataType=FLOAT)
      Arg (ref=BLOCKING, DataType=FLOAT)
  SynchActions:
    SABlocks:
      default (IsDefault=Yes)
        cyclic (Inline=Yes)
          Arg (ref=ACTIONS, DataType=STATEMENTS)
          Arg (ref=ID, DataType=FLOAT, DefaultInt=-1, MinCount=0, MaxCount=1)
      whenever:
        cyclic (Inline=Yes)
          Arg (ref=COND, DataType=FLOAT)
          Arg (ref=ACTIONS, DataType=STATEMENTS)
          Arg (ref=ID, DataType=FLOAT, DefaultInt=-1, MinCount=0, MaxCount=1)
      when:
        cyclic (Inline=Yes)
          Arg (ref=COND, DataType=FLOAT)
          Arg (ref=ACTIONS, DataType=STATEMENTS)
          Arg (ref=ID, DataType=FLOAT, DefaultInt=-1, MinCount=0, MaxCount=1)
      every:
        cyclic (Inline=Yes)
          Arg (ref=COND, DataType=FLOAT)
          Arg (ref=ACTIONS, DataType=STATEMENTS)
          Arg (ref=ID, DataType=FLOAT, DefaultInt=-1, MinCount=0, MaxCount=1)
      from:
        cyclic (Inline=Yes)
          Arg (ref=COND, DataType=FLOAT)
          Arg (ref=ACTIONS, DataType=STATEMENTS)
          Arg (ref=ID, DataType=FLOAT, DefaultInt=-1, MinCount=0, MaxCount=1)
    NonModalActivation:
      Start = @#thread.sa_last_keep_alive = 1;
        ActivateCyclicGroup(:-1:);
      Stop = WaitStopCyclicGroups(:(:-1:):);
  ParserData (NestedComments=Yes, DefaultCaseSensitive=No, CommentsSpanLines=No, SubDeclsLocalToFile=Yes, ProgDeclsLocalToFile=Yes, AllowUnprefixedFileCalls=Yes, AllowUnprefixedSubCalls=Yes, LocalVarScopeForMainProg=No, FileScopeVarsVisibleInSub=Yes, MainPrgReturnAtNextMainPrgHdr=Yes, AllowVarReadBeforeAssign=No, AllowArrayRefWithoutIndex=Yes, AllowNamedFnArgs=Yes, AllowBuiltinFnArgsOutOfSequence=Yes, AllowBuiltInProcCallWithoutBrackets=Yes, AllowBuiltInFnCallWithoutBrackets=No, AllowPLCFnCallWithoutBrackets=No, AllowStructMemberAutoDereference=Yes, AllowVariableAutoDereference=Yes, EnableStringCharacterIndexing=Yes, AllowIgnoredExtraSubArgs=Yes, OnMacroRedefinition=Error, CheckFileTimestampBeforeCalls=Yes)
    TKG_END_OF_LINE = \n (IsPattern=No)
    TKG_LINE_CONTINUE = \ (IsPattern=No, FileXLInvalid=Yes)
    TKG_LINE_BREAK = @@
    TKG_OPEN_COMMENT = ;
    TKG_CLOSE_COMMENT
    TKG_TRUE = TRUE:\W (IsPattern=Yes)
    TKG_FALSE = FALSE:\W (IsPattern=Yes)
    TKG_PAREVAL_MODAL_ID = ID:[\s=] (FileXLInvalid=Yes, IsPattern=Yes)
    TKG_MACRO_DEFINE_GLOBAL = define\s+ip_global:\s (IsPattern=Yes, FollowedBy=TKG_MACRO_NAME)
    TKG_MACRO_DEFINE = define\s+local:\s|define:\s (IsPattern=Yes, FollowedBy=TKG_MACRO_NAME)
    TKG_MACRO_UNDEFINE = undefine:\s (IsPattern=Yes, FollowedBy=TKG_MACRO_NAME)
    TKG_MACRO_AS = as:[\s\n] (IsPattern=Yes, FollowedBy=TKG_MACRO_TEXT)
    TKG_PROG_START = %:[^L] (IsPattern=Yes, CaseSensitive=Yes, FollowedBy=TKG_PROG_NAME)
    TKG_PROG_NAME = [\w\d]+ (IsPattern=Yes, Restricted=Yes)
    TKG_SET_MODAL_SUB = MCALL:\W (FileXLInvalid=Yes, IsPattern=Yes)
    TKG_INDIR_PROG_CALL = CALL:\s (IsPattern=Yes)
    TKG_INDIR_PROG_BLOCK = BLOCK:\s (FileXLInvalid=Yes, IsPattern=Yes)
    TKG_PROC_START = PROC:\s (FileXLInvalid=Yes, IsPattern=Yes, FollowedBy=TKG_PROC_NAME)
    TKG_PROC_NAME = \w[\w\d]+ (IsPattern=Yes, Restricted=Yes)
    TKG_ARG_PASSBYREF = VAR:\s (IsPattern=Yes)
    TKG_SUBPROG_PROTO = INTERN:\s (IsPattern=Yes, FollowedBy=TKG_SUBPROG_NAME)
    TKG_SUBPROG_START = SUB\s|%:L (FileXLInvalid=Yes, IsPattern=Yes, CaseSensitive=Yes, FollowedBy=TKG_SUBPROG_NAME)
    TKG_SUBPROG_NAME = \w[\w\d]+ (IsPattern=Yes, Restricted=Yes)
    TKG_EXTERN = EXTERN:\s (IsPattern=Yes, FollowedBy=TKG_PROG_FILE_NAME)
    TKG_PROG_FILE_NAME = [\^#&@']?[\w\d\./\:]+ (IsPattern=Yes, Restricted=Yes)
    TKG_PV_DECL = def:\s (IsPattern=Yes)
    TKG_PV_UNDECL = ~def:\s (IsPattern=Yes)
    TKG_VAR_RETAIN = retain:\s (IsPattern=Yes)
    TKG_VARSCOPE_IP_LOCAL = local:[\s\n] (IsPattern=Yes)
    TKG_VARSCOPE_IP_GLOBAL = ip_global:[\s\n] (IsPattern=Yes)
    TKG_VARSCOPE_NC_GLOBAL = nc_global:[\s\n] (IsPattern=Yes)
    TKG_VARSCOPE_PLC_GLOBAL = plc_global:[\s\n] (IsPattern=Yes)
    TKG_VARSYNCH_IP = ip_synch:\s (IsPattern=Yes)
    TKG_VARSYNCH_PATH = path_synch:\s (IsPattern=Yes)
    TKG_PAREVAL_DO = do:\s (FileXLInvalid=Yes, IsPattern=Yes)
    TKG_GOTOF = gotof:\s (FileXLInvalid=Yes, IsPattern=Yes, OptFollowedBy=TKG_GOTO_DEST)
    TKG_GOTOB = gotob:\s (FileXLInvalid=Yes, IsPattern=Yes, OptFollowedBy=TKG_GOTO_DEST)
    TKG_GOTO = goto:\s (FileXLInvalid=Yes, IsPattern=Yes, OptFollowedBy=TKG_GOTO_DEST)
    TKG_GOTO_DEST = \w[\w\d]* (IsPattern=Yes, Restricted=Yes)
    TKG_ARITH_BINARY_INT_DIVIDE = DIV:[\s(] (IsPattern=Yes)
    TKG_ARITH_BINARY_MODULO = MOD:[\s(] (IsPattern=Yes)
    TKG_FOR = FOR:\s (FileXLInvalid=Yes, IsPattern=Yes)
    TKG_ENDFOR = ENDFOR:[\s\n] (FileXLInvalid=Yes, IsPattern=Yes)
    TKG_FORTO = TO:\W (IsPattern=Yes)
    TKG_DO = repeat:[\s\n] (FileXLInvalid=Yes, IsPattern=Yes)
    TKG_ENDDO_UNTIL = until:[\s(] (FileXLInvalid=Yes, IsPattern=Yes)
    TKG_LOGICAL_UNARY_NOT = not:\W (IsPattern=Yes)
    TKG_SUPPRESS_SINGLE_STEP = NOHALT
    TKG_NC_BLOCK_PREFIX = N:[\s\d] (IsPattern=Yes)
    TKG_LOGICAL_HP_BINARY_AND = and:\W (IsPattern=Yes)
    TKG_LOGICAL_HP_BINARY_OR = or:\W (IsPattern=Yes)
    TKG_LOGICAL_HP_BINARY_XOR = xor:\W (IsPattern=Yes)
    TKG_BITWISE_BINARY_AND = b_and:\W (IsPattern=Yes)
    TKG_BITWISE_BINARY_OR = b_or:\W (IsPattern=Yes)
    TKG_BITWISE_BINARY_XOR = b_xor:\W (IsPattern=Yes)
    TKG_BITWISE_UNARY_COMPLEMENT = b_not:\W (IsPattern=Yes)
    TKG_PATHSYNCH_REC_IEC = do_path_synch:\W (FileXLInvalid=Yes, IsPattern=Yes)
    TKG_PATHSYNCH_END = end_path_synch:\W (FileXLInvalid=Yes, IsPattern=Yes)
    TKG_PATHSYNCH_IPEVAL = ip_eval:\W (FileXLInvalid=Yes, IsPattern=Yes)
    TKG_IF = if:\W (FileXLInvalid=Yes, IsPattern=Yes)
    TKG_THEN = then:\W (FileXLInvalid=Yes, IsPattern=Yes)
    TKG_BLOCK_ELSE = else:\W (FileXLInvalid=Yes, IsPattern=Yes)
    TKG_BLOCK_ENDIF = endif:\W (FileXLInvalid=Yes, IsPattern=Yes)
    TKG_SWITCH = case:\W (FileXLInvalid=Yes, IsPattern=Yes)
    TKG_SWITCH_OF = of:\W (FileXLInvalid=Yes, IsPattern=Yes)
    TKG_SWITCH_DEFAULT = default:\W (FileXLInvalid=Yes, IsPattern=Yes)
    TKG_WHILE = while:\W (FileXLInvalid=Yes, IsPattern=Yes)
    TKG_ENDWHILE = endwhile (FileXLInvalid=Yes)
    TKG_FOREVER = loop:\W (FileXLInvalid=Yes, IsPattern=Yes)
    TKG_ENDFOREVER = endloop:\W (FileXLInvalid=Yes, IsPattern=Yes)
    TKG_LABEL_DEF = \w:\:|\w[\w\d]+:\: (IsPattern=Yes, FollowedBy=TKG_LABEL_SUFFIX)
    TKG_LABEL_SUFFIX = : (Restricted=Yes)
    TKG_MACRO_TEXT = . (Restricted=Yes, IsPattern=Yes)
    TKG_MACRO_NAME = [$\w][$\w\d(]+ (Restricted=Yes, IsPattern=Yes)
    TKG_PRIM_TYPE (IsPattern=Yes)
    TKG_OPEN_BRACKET = (
    TKG_CLOSE_BRACKET = )
    TKG_OPEN_INDEXBRACKET = [
    TKG_CLOSE_INDEXBRACKET = ]
    TKG_COMMA = ,
    TKG_DOT = \.:\w (IsPattern=Yes, FollowedBy=TKG_STRUCT_MEMBER_REF)
    TKG_STRUCT_MEMBER_REF = \w|\w[\w\d]+ (IsPattern=Yes, Restricted=Yes)
    TKG_PARAM_PREFIX = R:[\[\d]|$[RP]:[\[\d]|M[WLF]:[\[\d]|EX[WLBF]:[\[\d] (IsPattern=Yes)
    TKG_SUBRANGE = ..
    TKG_NUMBER = \d+\.\d+|\d+\.:[^\.] (IsPattern=Yes)
    TKG_INTEGER = \d+ (IsPattern=Yes)
    TKG_FRACTION = \.\d+ (IsPattern=Yes)
    TKG_NUMBER_EXP = EX:[\s\d\+\-\.] (IsPattern=Yes)
    TKG_STRING_CONCAT = <<
    TKG_COMP_BINARY_GREATER_THAN_OR_EQ = >=
    TKG_COMP_BINARY_LESS_THAN_OR_EQ = <=
    TKG_COMP_BINARY_EQUAL_TO = ==
    TKG_COMP_BINARY_NOT_EQUAL_TO = <>
    TKG_COMP_BINARY_GREATER_THAN = >
    TKG_COMP_BINARY_LESS_THAN = <
    TKG_ASSIGN_INCR = =ic:( (IsPattern=Yes)
    TKG_ASSIGN_EQ = =
    TKG_ARITH_BINARY_PLUS = +
    TKG_ARITH_BINARY_MINUS = -
    TKG_ARITH_BINARY_MULTIPLY = *
    TKG_ARITH_BINARY_DIVIDE = /
    TKG_SUBCALL_REPEAT_PREFIX = P:[\s\d] (IsPattern=Yes, FollowedBy=TKG_INTEGER)
    TKG_PV_DECL_REF = \w[\w\d\.\:\*]* (IsPattern=Yes, Restricted=Yes)
    TKG_G_CODE_PREFIX = G:[\s\d] (IsPattern=Yes)
    TKG_M_CODE_PREFIX = M:[\s\d(] (IsPattern=Yes)
    TKG_FUB_DECL = fub\s (IsPattern=Yes)
    TKG_FUB_ERR_LEV_1 = error_level_1:\s (IsPattern=Yes)
    TKG_FUB_ERR_LEV_2 = error_level_2:\s (IsPattern=Yes)
    TKG_FUB_ERR_LEV_3 = error_level_3:\s (IsPattern=Yes)
    TKG_FUB_ERR_LEV_4 = error_level_4:\s (IsPattern=Yes)
    TKG_FUB_BLOCKING = blocking:[\s\n] (IsPattern=Yes)
    TKG_FUB_NON_BLOCKING = non_blocking:\s (IsPattern=Yes)
    TKG_IEC_TYPED_VALUE = #[\w\d]+:[^\w\d\:] (IsPattern=Yes)
    TKG_REFERENCE = ref:[\s\n]|reference:[\s\n] (IsPattern=Yes, FollowedBy=TKG_IEC_TO)
    TKG_IEC_TO = to:[\s\n] (IsPattern=Yes, Restricted=Yes)
    TKG_ACCESS = ACCESS:[\s\n] (IsPattern=Yes)
    TKG_BINARY_LITERAL_START = 'B:[01_] (FollowedBy=TKG_BINARY_LITERAL_BODY, IsPattern=Yes)
    TKG_BINARY_LITERAL_BODY = [01_]+' (Restricted=Yes, IsPattern=Yes)
    TKG_HEX_LITERAL_START = 'H:[\dA-F_] (FollowedBy=TKG_HEX_LITERAL_BODY, IsPattern=Yes)
    TKG_HEX_LITERAL_BODY = [\dA-F_]+' (Restricted=Yes, IsPattern=Yes)
    TKG_WORD = \w|\w[\w\d\./]+|\./\w|\./\w[\w\d\./]+|[\^#][\w\d]+\:[\w\d\./]+ (IsPattern=Yes)
  StringChars (AsciiStringStart=", AsciiStringEnd=", UTF16StringStart=W", UTF16StringEnd=")
    EscapeSeq (Search=$N, ReplaceValue=10)
    EscapeSeq (Search=$L, ReplaceValue=10)
    EscapeSeq (Search=$P, ReplaceValue=12)
    EscapeSeq (Search=$R, ReplaceValue=13)
    EscapeSeq (Search=$T, ReplaceValue=9)
    EscapeSeq (Search=$Q, ReplaceStr=")
    EscapeSeq (Search=$', ReplaceStr=')
    EscapeSeq (Search=$", ReplaceStr=")
    EscapeSeq (Search=$[\dA-Fa-f]+, IsPattern=Yes, ReplaceEncodingBase=16)
    EscapeSeq (Search=$$, ReplaceStr=$)
    EscapeSeq (Search=$, ReplaceStr=)
```

### Data object Logical/GmcIpConfig/gmcipcsm (Cnc, version 5.02.1)

#### gmcipcsm.cnc
```
Root (LangModule=ailgcode, Version=1.0)
  Constants:
    NumAxes = 15 (Type=INT)
  Preprocess:
    PP_RULE_STOPRE (Search=STOPRE, Replace=G172)
    PP_RULE_CIP (Search=CIP:\W, Replace=G102, IsPattern=Yes)
  Types:
    RotationAngleSpecifier (type=ENUM, EnumType=REGEXP, Value6=H)
    RadiusSpecifier (type=ENUM, EnumType=REGEXP, Value1=R\s*=, Value2=CR\s*=)
    InterpolParam (type=ENUM, EnumType=REGEXP, Value0=I, Value1=J, Value2=K, Value100=G161\s*I, Value101=G161\s*J, Value102=G161\s*K, Value200=G162\s*I, Value201=G162\s*J, Value202=G162\s*K, Value0300=I\s*=\s*AC, Value0301=J\s*=\s*AC, Value0302=K\s*=\s*AC, Value0400=I\s*=\s*IC, Value0401=J\s*=\s*IC, Value0402=K\s*=\s*IC)
    CirclePointParam (type=ENUM, EnumType=REGEXP, Value0=I1\s*=, Value1=J1\s*=, Value2=K1\s*=, Value100=G161\s*I1\s*=, Value101=G161\s*J1\s*=, Value102=G161\s*K1\s*=, Value200=G162\s*I1\s*=, Value201=G162\s*J1\s*=, Value202=G162\s*K1\s*=, Value0300=I1\s*=\s*AC, Value0301=J1\s*=\s*AC, Value0302=K1\s*=\s*AC, Value0400=I1\s*=\s*IC, Value0401=J1\s*=\s*IC, Value0402=K1\s*=\s*IC)
    RPYAngleName (type=ENUM, EnumType=REGEXP, Value1=ROLL, Value0=PITCH, Value2=YAW)
    EulerAngleName (type=ENUM, EnumType=REGEXP, Value3=PHI, Value4=THETA, Value5=PSI)
    RotaryVectorName (type=ENUM, EnumType=REGEXP, Value0=P\s*=, Value1=Q\s*=, Value2=R\s*=)
    DwellTime (type=FLOAT)
    RParamIndex (type=INT, MinValue=0, MaxValue=999)
    EXParamIndex (type=INT, MinValue=0, MaxValue=99)
    MParamIndex (type=INT, MinValue=0, MaxValue=99)
    Byte (type=INT, MinValue=0, MaxValue=255)
    Word (type=INT, MinValue=-32768, MaxValue=32767)
    Long (type=INT)
  PVMacros:
    SAVE (ArrayDims=0, Group=500)
      CALL = Info(:id:52101, msg:"Save Modal GCode State NOT SUPPORTED YET":);
  SysVars
  Parameters:
    R (IndexType=RParamIndex, ValueType=FLOAT)
      ARG (ref=EXPR, DataType=RParamIndex)
    QUOTED (QuotedName=$R, Synchronous=Yes, IndexType=RParamIndex, ValueType=FLOAT)
      ARG (ref=EXPR, DataType=RParamIndex)
    QUOTED (QuotedName=$P, Synchronous=Yes, IndexType=RParamIndex, ValueType=FLOAT)
      ARG (ref=EXPR, DataType=RParamIndex)
    EXB (IndexType=EXParamIndex, ValueType=Byte)
      ARG (ref=EXPR, DataType=EXParamIndex)
    EXW (IndexType=EXParamIndex, ValueType=Word)
      ARG (ref=EXPR, DataType=EXParamIndex)
    EXL (IndexType=EXParamIndex, ValueType=Long)
      ARG (ref=EXPR, DataType=EXParamIndex)
    EXF (IndexType=EXFParamIndex, ValueType=FLOAT)
      ARG (ref=EXPR, DataType=EXFParamIndex)
    MW (Synchronous=Yes, IndexType=MParamIndex, ValueType=Word)
      ARG (ref=EXPR, DataType=MParamIndex)
    ML (Synchronous=Yes, IndexType=MParamIndex, ValueType=Long)
      ARG (ref=EXPR, DataType=MParamIndex)
    MF (Synchronous=Yes, IndexType=MParamIndex, ValueType=FLOAT)
      ARG (ref=EXPR, DataType=MParamIndex)
  MCodes:
    M17 = 17 (Group=41, Alias=RET:[^\d\w\(], Eval=Early, Inline=Yes, AliasIsPattern=Yes)
      ARG (ref=VALUE, DataType=FLOAT, RequireLiteral=Yes)
    M17_1 = 17.1 (Group=41, Alias=CONDRET, Eval=Early, Inline=Yes)
      ARG (ref=VALUE, DataType=FLOAT, RequireLiteral=Yes)
```

### Data object Logical/GmcIpConfig/gmcipcfg (Cnc, version 5.02.1)

#### gmcipcfg.cnc
```
CONFIG:
  LANG_INCLUDE gmcipmxd (LangName=IEC-ST, DataObject=Yes, IfNotExist=Error, Scope=NC_GLOBAL, RequireFnIgnore=MXConvertOrient)
  XML_INCLUDE gmcipvar (IfNotExist=Warn)
  XML_INCLUDE gmcipfun (IfNotExist=Warn)
  XML_INCLUDE gmcipfub (IfNotExist=Warn)
  MPQUEUE (NumPackets=200, LookaheadMinBlocks=5, LookaheadMaxBlocks=20, LookaheadMode=any, MaxPathJobs=256, CheckForNaNs=1)
  MONITOR (MaxPathStackEvents=1024)
  MPLOG (MaxBuffers=10, MinBuffers=4, EarlyCircleBufferLookahead=2, DefaultBufferSize=131072, TaskCycleDelay=1, FileDevice=mplog*, MaxLogFiles=20, MaxLogFileSize=1048576, CopyLineTextMaxChars=80)
  AXES (StandardCNCAxes=Yes)
  FUBOutputs:
    FUBOutput PLCOpen:
      ERROR (condition=$Error == 1)
      BUSY (condition=$Busy == 1)
    FUBOutput BuR:
      ERROR (condition=$status != 65535 && $status != 0)
      BUSY (condition=$status == 65535)
  FUNCTIONS:
    FUNC LEN (DeclareName=__LEN, AlwaysDeclare=Yes, RetType=INT)
      ARG IN (Type=STRING)
    FUNC LEFT (DeclareName=__LEFT, AlwaysDeclare=Yes, RetType=STRING, RetRef=Yes)
      ARG IN (Type=STRING)
      ARG L (Type=INT)
    FUNC RIGHT (DeclareName=__RIGHT, AlwaysDeclare=Yes, RetType=STRING, RetRef=Yes)
      ARG IN (Type=STRING)
      ARG L (Type=INT)
    FUNC MID (DeclareName=__MID, AlwaysDeclare=Yes, RetType=STRING, RetRef=Yes)
      ARG IN (Type=STRING)
      ARG L (Type=INT)
      ARG P (Type=INT)
    FUNC CONCAT (DeclareName=__CONCAT, AlwaysDeclare=Yes, RetType=STRING, RetRef=Yes)
      ARG IN1 (Type=STRING)
      ARG IN2 (Type=STRING)
    FUNC INSERT (DeclareName=__INSERT, AlwaysDeclare=Yes, RetType=STRING, RetRef=Yes)
      ARG IN1 (Type=STRING)
      ARG IN2 (Type=STRING)
      ARG P (Type=INT)
    FUNC DELETE (DeclareName=__DELETE, AlwaysDeclare=Yes, RetType=STRING, RetRef=Yes)
      ARG IN (Type=STRING)
      ARG L (Type=INT)
      ARG P (Type=INT)
    FUNC REPLACE (DeclareName=__REPLACE, AlwaysDeclare=Yes, RetType=STRING, RetRef=Yes)
      ARG IN1 (Type=STRING)
      ARG IN2 (Type=STRING)
      ARG L (Type=INT)
      ARG P (Type=INT)
    FUNC FIND (DeclareName=__FIND, AlwaysDeclare=Yes, RetType=INT)
      ARG IN1 (Type=STRING)
      ARG IN2 (Type=STRING)
  XML_INCLUDE gmcipuc (IfNotExist=Warn)
```

### Data object Logical/GmcIpConfig/gmcipiec (Cnc, version 5.02.1)
